// ---- BECKHOFF SPECIFIC helper library/POUs/MethodCall/UA_MethodCall_ADSReadWriteReq.TcPOU
FUNCTION_BLOCK UA_MethodCall_ADSReadWriteReq
VAR_INPUT
	bExecute			: BOOL;
	nConnectionHdl		: DWORD;
	nNamespaceIndex		: UINT; 			(* to be retrieved using UA_GetNamespaceIndex *)
	sNetID				: T_AmsNetId; 		(* AmsNetId OF the Target *)
	nPort				: INT; 			(* Port number	*)
	nIndexGroup			: DINT;			(* IndexGroup*)
	nIndexOffset		: DINT; 			(* IndexOffset*)
	pWriteData			: PVOID;
	cbWriteData			: UDINT;			(* Count of bytes to be read*)
	pReadArgInfoAndData	: PVOID;
	cbReadArgInfoAndData: UDINT;			(* Count of bytes to be read*)
	nNumberOfOutputArguments	: UDINT; 
	pOutputArgInfo		: POINTER TO ST_UAMethodArgInfo; 
	cbOutputArgInfo		: UDINT;
	Timeout				: TIME := DEFAULT_ADS_TIMEOUT;
END_VAR
VAR_OUTPUT
	cbReadData_R		: UDINT;
	bDone				: BOOL;
	bBusy				: BOOL;
	bError				: BOOL;
	nErrorID			: DWORD;
END_VAR
VAR
	iRdWrtReqState		: INT;
	RTrig				: R_TRIG;

	fbUA_MethodGetHandle: UA_MethodGetHandle;
	nMethodHdl			: DWORD;
	ObjectNodeID		: ST_UANodeID;
	MethodNodeID		: ST_UANodeID;

	fbUA_MethodCall		: UA_MethodCall;
	InputArguments		: ARRAY [1..nNumberOfInputArguments] OF ST_UAMethodArgInfo; (*ReadWriteReq has 6 input parameters *)	
	nArg				: INT;
	nInputData			: ARRAY [1..nInputArgSize] OF BYTE; // (* NetID(24)+ Port(2)+ IG(4)+ IO(4)*)
	nOffset				: UDINT;

	fbUA_MethodReleaseHandle	: UA_MethodReleaseHandle;
	bInputDataError				: BOOL; 
END_VAR
VAR CONSTANT
	nInputArgSize			: UDINT := 34; // (* NetID(24)+ Port(2)+ IG(4)+ IO(4)*)
	nNumberOfInputArguments : UDINT := 6;
END_VAR

(*
ADSReadWriteReq(
******** Input Arguments ********
	string sNetID, 		: AmsNetId of the Target
	int16 Port,			: Port number	
	int32 IndexGroup,		: IndexGroup
	int32 IndexOffset,		: IndexOffset
	ByteString WriteData	: Data to be written to the device
	uint32 cbReadData		: Count of bytes to be read
******** Output Arguments ********
	bytestring Data		: count of bytes actually read
);
*)

RTrig(CLK:= bExecute);

CASE iRdWrtReqState OF

0:	(* Get Method Handle *)
	IF RTrig.Q THEN
		bBusy		:= TRUE;
		bDone 		:= FALSE;
		bError		:= FALSE;
		nErrorID	:= 0;
		ObjectNodeID.eIdentifierType 	:= eUAIdentifierType_String;
		ObjectNodeID.nNamespaceIndex 	:= nNamespaceIndex;
		ObjectNodeID.sIdentifier		:= 'ADSAMS';
	
		MethodNodeID.eIdentifierType 	:= eUAIdentifierType_String;
		MethodNodeID.nNamespaceIndex 	:= nNamespaceIndex;
		MethodNodeID.sIdentifier		:= 'ADSAMS.AdsReadWriteReq';

		M_Init();
		IF bInputDataError = FALSE THEN
			iRdWrtReqState 	:= iRdWrtReqState + 1;
		ELSE
			bBusy		:= FALSE; 
			bError 		:= TRUE;
			nErrorID 	:= DEVICE_INVALIDSIZE; //16#705 parameter size not correct
		END_IF
	END_IF


1:	(* Method Get Handle *)
	fbUA_MethodGetHandle(
			Execute			:= TRUE,
			ConnectionHdl	:= nConnectionHdl,
			ObjectNodeID	:= ObjectNodeID,
			MethodNodeID 	:= MethodNodeID,
			Timeout			:= Timeout,
			MethodHdl		=> nMethodHdl
		);
	IF NOT fbUA_MethodGetHandle.Busy THEN
		fbUA_MethodGetHandle(Execute := FALSE);

		IF NOT fbUA_MethodGetHandle.Error THEN
			(*  *)
			iRdWrtReqState := iRdWrtReqState + 1; (* Call Method *)
		ELSE
			bError			:= TRUE;
			nErrorID		:= fbUA_MethodGetHandle.ErrorID;
			iRdWrtReqState := 3; (* Release Handle *)
		END_IF
	END_IF


2:	(* Method Call *)
	fbUA_MethodCall(
		Execute					:= TRUE,
		ConnectionHdl			:= nConnectionHdl,
		MethodHdl				:= nMethodHdl,
		nNumberOfInputArguments := nNumberOfInputArguments,		(* 6 *)
		pInputArgInfo			:= ADR(InputArguments),
		cbInputArgInfo			:= SIZEOF(InputArguments),
		pInputArgData			:= ADR(nInputData),
		cbInputArgData			:= nOffset,
		pInputWriteData			:= pWriteData,
		cbInputWriteData		:= cbWriteData,
		nNumberOfOutputArguments:= nNumberOfOutputArguments,		(* 6 *)
		pOutputArgInfo			:= pOutputArgInfo,
		cbOutputArgInfo			:= cbOutputArgInfo,
		pOutputArgInfoAndData	:= pReadArgInfoAndData,
		cbOutputArgInfoAndData	:= cbReadArgInfoAndData,
		Timeout					:= Timeout
	);
	IF NOT fbUA_MethodCall.Busy THEN
		fbUA_MethodCall(Execute := FALSE, cbRead_R => cbReadData_R);

		IF NOT fbUA_MethodCall.Error THEN
			(*  *)
			iRdWrtReqState 	:= iRdWrtReqState + 1; (* Release handle *)
		ELSE
			bError			:= TRUE;
			nErrorID		:= fbUA_MethodCall.ErrorID;
			iRdWrtReqState	:= 3; (* Release handle *)
		END_IF
	END_IF


3:	(* Release Method Handle *)
	fbUA_MethodReleaseHandle(
		Execute			:= TRUE,
		ConnectionHdl	:= nConnectionHdl,
		MethodHdl		:= nMethodHdl,
		Timeout			:= Timeout
	);

	IF NOT fbUA_MethodReleaseHandle.Busy THEN
		fbUA_MethodReleaseHandle(Execute := FALSE);
		bBusy := FALSE;
		IF NOT fbUA_MethodReleaseHandle.Error THEN
			(* session closed *)
			bDone := TRUE;
			iRdWrtReqState 	:= 0; (* idle *)
		ELSE
			bError		:= TRUE;
			nErrorID		:= fbUA_MethodReleaseHandle.ErrorID;
			iRdWrtReqState 	:= 0; (* idle *)
		END_IF
	END_IF
END_CASE

ACTION M_Init:
bInputDataError := FALSE; 
nOffset := 0;
MEMSET(ADR(InputArguments),0,SIZEOF(InputArguments));
MEMSET(ADR(nInputData),0,SIZEOF(nInputData));

nArg := 1;
(*sNetID := sAmsNetID;*)	(********** NET ID **********)
InputArguments[nArg].DataType			:= eUAType_String;
InputArguments[nArg].ValueRank			:= -1; 							(* Scalar = -1 or Array *)
InputArguments[nArg].ArrayDimensions[1]	:= 0; 							(* Number of Dimension in case its an array *)
InputArguments[nArg].nLenData			:= INT_TO_UDINT(LEN(sNetId)) + 1;				(* Length if its a STRING *)
IF nOffset + INT_TO_UDINT(LEN(sNetId))+1 > nInputArgSize THEN 
	bInputDataError := TRUE;
	RETURN;
ELSE
	MEMCPY(ADR(nInputData)+nOffset,ADR(sNetId),INT_TO_UDINT(LEN(sNetId))+1);				(* VALUE in BYTES FORM *)
	nOffset := nOffset + INT_TO_UDINT(LEN(sNetId))+1;
END_IF

nArg := nArg + 1;
(* nPort := 851;*)			(********** PORT **********)
InputArguments[nArg].DataType			:= eUAType_Int16;
InputArguments[nArg].ValueRank			:= -1; 							(* Scalar = -1 or Array *)
InputArguments[nArg].ArrayDimensions[1]	:= 0; 							(* Number of Dimension in case its an array *)
InputArguments[nArg].nLenData			:= SIZEOF(nPort);				(* Length if its a STRING *)
IF nOffset + SIZEOF(nPort) > nInputArgSize THEN 
	bInputDataError := TRUE;
	RETURN;
ELSE
	MEMCPY(ADR(nInputData)+nOffset,ADR(nPort),SIZEOF(nPort));			(* VALUE in BYTES FORM *)
	nOffset := nOffset + SIZEOF(nPort);
END_IF

nArg := nArg + 1;
(*nIndexGroup := 16#4020;*)	(********** INDEX GROUP **********)
InputArguments[nArg].DataType			:= eUAType_Int32;
InputArguments[nArg].ValueRank			:= -1; 							(* Scalar = -1 or Array *)
InputArguments[nArg].ArrayDimensions[1]	:= 0; 							(* Number of Dimension in case its an array *)
InputArguments[nArg].nLenData			:= SIZEOF(nIndexGroup);			(* Length if its a STRING *)
IF nOffset + SIZEOF(nIndexGroup) > nInputArgSize THEN 
	bInputDataError := TRUE;
	RETURN;
ELSE
	MEMCPY(ADR(nInputData)+nOffset,ADR(nIndexGroup),SIZEOF(nIndexGroup));		(* VALUE in BYTES FORM *)
	nOffset := nOffset + SIZEOF(nIndexGroup);
END_IF

nArg := nArg + 1;
(*nIndexOffset := 0; *)		(********** INDEX OFFSET **********)
InputArguments[nArg].DataType			:= eUAType_Int32;
InputArguments[nArg].ValueRank			:= -1; 							(* Scalar = -1 or Array *)
InputArguments[nArg].ArrayDimensions[1]	:= 0; 							(* Number of Dimension in case its an array *)
InputArguments[nArg].nLenData			:= SIZEOF(nIndexOffset);		(* Length if its a STRING *)
IF nOffset + SIZEOF(nIndexOffset) > nInputArgSize THEN 
	bInputDataError := TRUE;
	RETURN;
ELSE
	MEMCPY(ADR(nInputData)+nOffset,ADR(nIndexOffset),SIZEOF(nIndexOffset));	(* VALUE in BYTES FORM *)
	nOffset := nOffset + SIZEOF(nIndexOffset);
END_IF

nArg := nArg + 1;
(*Data := 2; *)		(*********** WriteData ***********)
InputArguments[nArg].DataType			:= eUAType_ByteString;
InputArguments[nArg].ValueRank			:= -1; 						(* Scalar = -1 or Array *)
InputArguments[nArg].ArrayDimensions[1]	:= 0; 						(* Number of Dimension in case its an array *)
InputArguments[nArg].nLenData			:= cbWriteData;				(* Length if its a STRING *)

nArg := nArg + 1;
(*Data := 2; *)		(*********** ReadData size ***********)
InputArguments[nArg].DataType			:= eUAType_UInt32;
InputArguments[nArg].ValueRank			:= -1; 						(* Scalar = -1 or Array *)
InputArguments[nArg].ArrayDimensions[1]	:= 0; 						(* Number of Dimension in case its an array *)
InputArguments[nArg].nLenData			:= SIZEOF(cbReadArgInfoAndData);		(* Length if its a STRING *)
END_ACTION

END_FUNCTION_BLOCK

// ---- POUs/PRG_READ_List_woConnectIdent.TcPOU
PROGRAM PRG_READ_List_woConnectIdent
VAR
	fbUA_Connect			: UA_Connect;
	SessionConnectInfo		: ST_UASessionConnectInfo;
	sOpcUA_URL				: STRING(MAX_STRING_LENGTH);
	nConnectionHdl			: DWORD;

	fbUA_GetNamespaceIndex 	: UA_GetNamespaceIndex;
	nNamespaceIndex			: UINT;
	fbUA_NodeGetHandleList	: UA_NodeGetHandleList;
	NodeIDs					: ARRAY [1..nMaxNodeIDsInList] OF ST_UANodeID;
	nNodeHdls				: ARRAY [1..nMaxNodeIDsInList] OF DWORD;

	fbUA_ReadList			: UA_ReadList; 
	stIndexRange			: ARRAY [1..nMaxIndexRange] OF ST_UAIndexRange;
	nIndexRangeCount		: UINT;
	stNodeAddInfo			: ARRAY [1..nMaxNodeIDsInList] OF ST_UANodeAdditionalInfo;
	stReadListData			: ST_ReadListData; // memory block must contain the Data[], NodeErrorIDs[], TimeStamps[] and cbData_R[]
	cbData					: ARRAY [1..nMaxNodeIDsInList] OF UDINT; (* Bytes to be actually Read *)
	cbData_R				: UDINT;
	cbDataTotal				: UDINT; 
	
	fbUA_NodeReleaseHandleList	: UA_NodeReleaseHandleList;

	fbUA_Disconnect		: UA_Disconnect;

	iState		: INT;
	bTest		: BOOL:= TRUE;
	bDone		: BOOL;
	bBusy		: BOOL;
	bError		: BOOL;
	nErrorID	: DWORD;
	
	nNodeIdx	: INT; 
END_VAR


CASE iState OF
0:	(* idle *)
	IF bTest THEN
		bTest		:= FALSE;
		bError		:= FALSE;
		nErrorID	:= 0;

		(* Parameterize *)
		sOpcUA_URL						:= 'opc.tcp://pujal-nb03:4840';	(* OpcUA Url of the device with ip address *)

		SessionConnectInfo.tConnectTimeout 		:= T#1S;
		SessionConnectInfo.tSessionTimeout 		:= T#1S;
		SessionConnectInfo.sApplicationName		:= '';
//		SessionConnectInfo.sApplicationUri 		:= '';
		SessionConnectInfo.eSecurityMode 		:= eUASecurityMsgMode_None;
		SessionConnectInfo.eSecurityPolicyUri 	:= eUASecurityPolicy_None;
		SessionConnectInfo.eTransportProfileUri := eUATransportProfileUri_UATcp;

(*		nIndexRange[1].nStartIndex := 0;
		nIndexRange[1].nEndIndex := 1;
		nIndexRange[1].bRangeAccess := TRUE; *)
		iState	:= iState + 1;
	END_IF

1:	(* open UA session *)
	fbUA_Connect(
		Execute				:= TRUE,
		ServerURL			:= sOpcUA_URL,
		SessionConnectInfo  := SessionConnectInfo,
		Timeout				:= T#5S,
		ConnectionHdl		=> nConnectionHdl
	);

	IF NOT fbUA_Connect.Busy THEN
		fbUA_Connect(Execute := FALSE);

		IF NOT fbUA_Connect.Error THEN
			(* session open *)
			iState := iState + 1;
		ELSE
			bError			:= TRUE;
			nErrorID		:= fbUA_Connect.ErrorID;
			nConnectionHdl	:= 0;
			iState 			:= 0; (* idle *)
		END_IF
	END_IF


2:	(* GetNS Index *)
	fbUA_GetNamespaceIndex(
		Execute			:= TRUE,
		ConnectionHdl	:= nConnectionHdl,
		NamespaceUri	:= 'PLC1',
		NamespaceIndex	=> nNamespaceIndex
	);

	IF NOT fbUA_GetNamespaceIndex.Busy THEN
		fbUA_GetNamespaceIndex(Execute := FALSE);
		IF NOT fbUA_GetNamespaceIndex.Error THEN
			(* session closed *)
			iState 		:= iState + 1; (* idle *)
		ELSE
			bError		:= TRUE;
			nErrorID	:= fbUA_GetNamespaceIndex.ErrorID;
			iState 		:= 6; (* idle *)
		END_IF
	END_IF


3:	(* Get Node Handle *)
//	stNodeAddInfo[1].nIndexRangeCount := nIndexRangeCount;
//	stNodeAddInfo[1].stIndexRange := stIndexRange;
//	stNodeAddInfo[2].nIndexRangeCount := nIndexRangeCount;
//	stNodeAddInfo[2].stIndexRange := stIndexRange;
	nNodeIdx := 1;		//1
	
	NodeIDs[nNodeIdx].eIdentifierType := eUAIdentifierType_String;
	NodeIDs[nNodeIdx].nNamespaceIndex := nNamespaceIndex;
	NodeIDs[nNodeIdx].sIdentifier	:= 'MAIN.iVar1';
	
	nNodeIdx := nNodeIdx + 1; //2
	NodeIDs[nNodeIdx].eIdentifierType := eUAIdentifierType_String;
	NodeIDs[nNodeIdx].nNamespaceIndex := nNamespaceIndex;
	NodeIDs[nNodeIdx].sIdentifier	:= 'MAIN.diVar1';
	
	nNodeIdx := nNodeIdx + 1; //3
	NodeIDs[nNodeIdx].eIdentifierType := eUAIdentifierType_String;
	NodeIDs[nNodeIdx].nNamespaceIndex := nNamespaceIndex;
	NodeIDs[nNodeIdx].sIdentifier	:= 'MAIN.iVar2';
	
	nNodeIdx := nNodeIdx + 1; //4
	NodeIDs[nNodeIdx].eIdentifierType := eUAIdentifierType_String;
	NodeIDs[nNodeIdx].nNamespaceIndex := nNamespaceIndex;
	NodeIDs[nNodeIdx].sIdentifier	:= 'MAIN.diVar2';

	fbUA_NodeGetHandleList(
		Execute			:= TRUE,
		ConnectionHdl	:= nConnectionHdl,
		NodeIDCount 	:= gNodeIDCount, // 4
		NodeIDs			:= NodeIDs,
		NodeHdls		=> nNodeHdls
	);

	IF NOT fbUA_NodeGetHandleList.Busy THEN
		fbUA_NodeGetHandleList(Execute := FALSE);

		IF NOT fbUA_NodeGetHandleList.Error THEN
			(* session closed *)
			iState 		:= iState + 1; (* idle *)
		ELSE
			bError		:= TRUE;
			nErrorID	:= fbUA_NodeGetHandleList.ErrorID;
			iState 		:= 6; (* idle *)
		END_IF
	END_IF

	
4: 	(* UA_Read *)
	cbData[1] := SIZEOF(stReadListData.nIntVar1);
	cbData[2] := SIZEOF(stReadListData.nIntVar2);
	cbData[3] := SIZEOF(stReadListData.nIntVar3);
	cbData[4] := SIZEOF(stReadListData.nIntVar4);
	cbDataTotal := SIZEOF(stReadListData);
	fbUA_ReadList(
		Execute			:= TRUE,
		ConnectionHdl	:= nConnectionHdl,
		NodeHdlCount	:= gNodeIDCount, // 4
		NodeHdls		:= nNodeHdls,
		stNodeAddInfo 	:= stNodeAddInfo,
		pVariable		:= ADR(stReadListData),
		cbData			:= cbData ,
		cbDataTotal		:= cbDataTotal		
		);

	IF NOT fbUA_ReadList.Busy THEN
		fbUA_ReadList( Execute := FALSE, cbData_R => cbData_R);

		IF NOT fbUA_ReadList.Error THEN
			(* session closed *)
			iState 		:= iState + 1; (* idle *)
		ELSE
			bError		:= TRUE;
			nErrorID	:= fbUA_ReadList.ErrorID;
			iState 		:= 6; (* idle *)
		END_IF
	END_IF


5:	(* Release Node Handle *)
	fbUA_NodeReleaseHandleList(
		Execute			:= TRUE,
		ConnectionHdl	:= nConnectionHdl,
		NodeHdlCount	:= gNodeIDCount,	// 4
		NodeHdls		:= nNodeHdls
	);

	IF NOT fbUA_NodeReleaseHandleList.Busy THEN
		fbUA_NodeReleaseHandleList(Execute := FALSE);

		IF NOT fbUA_NodeReleaseHandleList.Error THEN
			(* session closed *)
			iState 		:= iState + 1; (* idle *)
		ELSE
			bError		:= TRUE;
			nErrorID	:= fbUA_NodeReleaseHandleList.ErrorID;
			iState 		:= 6; (* idle *)
		END_IF
	END_IF


6:	(* close session *)
	fbUA_Disconnect(
		Execute			:= TRUE,
		ConnectionHdl	:= nConnectionHdl
	);

	IF NOT fbUA_Disconnect.Busy THEN
		fbUA_Disconnect(Execute := FALSE);
		bBusy := FALSE;
		IF NOT fbUA_Disconnect.Error THEN
			(* session closed *)
			iState 		:= 0; (* idle *)
			IF NOT bError THEN 
				bDone 	:= TRUE;
			END_IF
		ELSE
			bError			:= TRUE;
			nErrorID		:= fbUA_Disconnect.ErrorID;
			iState 			:= 0; (* idle *)
			nConnectionHdl	:= 0;
		END_IF
	END_IF
END_CASE

END_PROGRAM

// ---- POUs/PRG_READ_List.TcPOU
PROGRAM PRG_READ_List
VAR
	fbUA_ConnectEx			: UA_Connect;
	SessionConnectInfoEx	: ST_UASessionConnectInfo;
	sOpcUA_URL				: STRING(MAX_STRING_LENGTH);
	nConnectionHdl			: DWORD;

	fbUA_GetNamespaceIndex 	: UA_GetNamespaceIndex;
	nNamespaceIndex			: UINT;
	fbUA_NodeGetHandleList	: UA_NodeGetHandleList;
	
	NodeIDs					: ARRAY [1..nMaxNodeIDsInList] OF ST_UANodeID;
	nNodeHdls				: ARRAY [1..nMaxNodeIDsInList] OF DWORD;

	fbUA_ReadList			: UA_ReadList;
	stIndexRange			: ARRAY [1..nMaxIndexRange] OF ST_UAIndexRange;
	nIndexRangeCount		: UINT;
	stNodeAddInfo			: ARRAY [1..nMaxNodeIDsInList] OF ST_UANodeAdditionalInfo;
	stReadListData			: ST_ReadListData; // memory block must contain the Data[], NodeErrorIDs[], TimeStamps[] and cbData_R[]
	cbData					: ARRAY [1..nMaxNodeIDsInList] OF UDINT; (* Bytes to be actually Read *)
	cbData_R				: UDINT;
	cbDataTotal				: UDINT; 
	
	fbUA_NodeReleaseHandleList	: UA_NodeReleaseHandleList;

	fbUA_Disconnect		: UA_Disconnect;

	iState		: INT;
	bTest		: BOOL:= TRUE;
	bDone		: BOOL;
	bBusy		: BOOL;
	bError		: BOOL;
	nErrorID	: DWORD;
	
	nNodeIdx	: INT; 
END_VAR


CASE iState OF
0:	(* idle *)
	IF bTest THEN
		bTest		:= FALSE;
		bError		:= FALSE;
		nErrorID	:= 0;

		(* Parameterize *)
		sOpcUA_URL						:= 'opc.tcp://pujal-nb03:4840';	(* OpcUA Url of the device with ip address *)

		SessionConnectInfoEx.tConnectTimeout 		:= T#5S;
		SessionConnectInfoEx.tSessionTimeout 		:= T#5S;
		SessionConnectInfoEx.sApplicationName		:= '';
		SessionConnectInfoEx.eSecurityMode 			:= eUASecurityMsgMode_None;
		SessionConnectInfoEx.eSecurityPolicyUri 	:= eUASecurityPolicy_None;
		SessionConnectInfoEx.eTransportProfileUri 	:= eUATransportProfileUri_UATcp;
		//SessionConnectInfoEx.stUserIdentTokenType

(*		nIndexRange[1].nStartIndex := 0;
		nIndexRange[1].nEndIndex := 1;
		nIndexRange[1].bRangeAccess := TRUE; *)
		iState	:= iState + 1;
	END_IF

1:	(* open UA session *)
	fbUA_ConnectEx(
		Execute				:= TRUE,
		ServerURL			:= sOpcUA_URL,
		SessionConnectInfo	:= SessionConnectInfoEx,
		Timeout				:= T#5S,
		ConnectionHdl		=> nConnectionHdl
	);

	IF NOT fbUA_ConnectEx.Busy THEN
		fbUA_ConnectEx(Execute := FALSE);

		IF NOT fbUA_ConnectEx.Error THEN
			(* session open *)
			iState := iState + 1;
		ELSE
			bError			:= TRUE;
			nErrorID		:= fbUA_ConnectEx.ErrorID;
			nConnectionHdl	:= 0;
			iState 			:= 0; (* idle *)
		END_IF
	END_IF


2:	(* GetNS Index *)
	fbUA_GetNamespaceIndex(
		Execute			:= TRUE,
		ConnectionHdl	:= nConnectionHdl,
		NamespaceUri	:= 'PLC1',
		NamespaceIndex	=> nNamespaceIndex
	);

	IF NOT fbUA_GetNamespaceIndex.Busy THEN
		fbUA_GetNamespaceIndex(Execute := FALSE);
		IF NOT fbUA_GetNamespaceIndex.Error THEN
			(* session closed *)
			iState 		:= iState + 1; (* idle *)
		ELSE
			bError		:= TRUE;
			nErrorID	:= fbUA_GetNamespaceIndex.ErrorID;
			iState 		:= 6; (* idle *)
		END_IF
	END_IF


3:	(* Get Node Handle *)
	nNodeIdx := 1;	
	NodeIDs[nNodeIdx].eIdentifierType := eUAIdentifierType_String;
	NodeIDs[nNodeIdx].nNamespaceIndex := nNamespaceIndex;
	NodeIDs[nNodeIdx].sIdentifier	:= 'MAIN.iVar1';
	cbData[nNodeIdx] := SIZEOF(stReadListData.nIntVar1);
	
	nNodeIdx := nNodeIdx + 1; 
	NodeIDs[nNodeIdx].eIdentifierType := eUAIdentifierType_String;
	NodeIDs[nNodeIdx].nNamespaceIndex := nNamespaceIndex;
	NodeIDs[nNodeIdx].sIdentifier	:= 'MAIN.iVar2';
	cbData[nNodeIdx] := SIZEOF(stReadListData.nIntVar2);
	
	nNodeIdx := nNodeIdx + 1; 	
	NodeIDs[nNodeIdx].eIdentifierType := eUAIdentifierType_String;
	NodeIDs[nNodeIdx].nNamespaceIndex := nNamespaceIndex;
	NodeIDs[nNodeIdx].sIdentifier	:= 'MAIN.iVar1';	
	cbData[nNodeIdx] := SIZEOF(stReadListData.nIntVar3);
	
	nNodeIdx := nNodeIdx + 1; 
	NodeIDs[nNodeIdx].eIdentifierType := eUAIdentifierType_String;
	NodeIDs[nNodeIdx].nNamespaceIndex := nNamespaceIndex;
	NodeIDs[nNodeIdx].sIdentifier	:= 'MAIN.iVar1';	
	cbData[nNodeIdx] := SIZEOF(stReadListData.nIntVar4);
	
	nNodeIdx := nNodeIdx + 1; 
	NodeIDs[nNodeIdx].eIdentifierType := eUAIdentifierType_String;
	NodeIDs[nNodeIdx].nNamespaceIndex := nNamespaceIndex;
	NodeIDs[nNodeIdx].sIdentifier	:= 'MAIN.iVar1';	
	cbData[nNodeIdx] := SIZEOF(stReadListData.nIntVar5);

	nNodeIdx := nNodeIdx + 1; 
	NodeIDs[nNodeIdx].eIdentifierType := eUAIdentifierType_String;
	NodeIDs[nNodeIdx].nNamespaceIndex := nNamespaceIndex;
	NodeIDs[nNodeIdx].sIdentifier	:= 'MAIN.iVar1';	
	cbData[nNodeIdx] := SIZEOF(stReadListData.nIntVar6);

	nNodeIdx := nNodeIdx + 1; 
	NodeIDs[nNodeIdx].eIdentifierType := eUAIdentifierType_String;
	NodeIDs[nNodeIdx].nNamespaceIndex := nNamespaceIndex;
	NodeIDs[nNodeIdx].sIdentifier	:= 'MAIN.iVar1';	
	cbData[nNodeIdx] := SIZEOF(stReadListData.nIntVar7);

	nNodeIdx := nNodeIdx + 1; 
	NodeIDs[nNodeIdx].eIdentifierType := eUAIdentifierType_String;
	NodeIDs[nNodeIdx].nNamespaceIndex := nNamespaceIndex;
	NodeIDs[nNodeIdx].sIdentifier	:= 'MAIN.iVar1';
	cbData[nNodeIdx] := SIZEOF(stReadListData.nIntVar8);	

	nNodeIdx := nNodeIdx + 1; 
	NodeIDs[nNodeIdx].eIdentifierType := eUAIdentifierType_String;
	NodeIDs[nNodeIdx].nNamespaceIndex := nNamespaceIndex;
	NodeIDs[nNodeIdx].sIdentifier	:= 'MAIN.iVar1';
	cbData[nNodeIdx] := SIZEOF(stReadListData.nIntVar9);

	nNodeIdx := nNodeIdx + 1; 
	NodeIDs[nNodeIdx].eIdentifierType := eUAIdentifierType_String;
	NodeIDs[nNodeIdx].nNamespaceIndex := nNamespaceIndex;
	NodeIDs[nNodeIdx].sIdentifier	:= 'MAIN.iVar1';
	cbData[nNodeIdx] := SIZEOF(stReadListData.nIntVar10);	

	cbDataTotal := SIZEOF(stReadListData);
	
	fbUA_NodeGetHandleList(
		Execute			:= TRUE,
		ConnectionHdl	:= nConnectionHdl,
		NodeIDCount 	:= gNodeIDCount, // 10
		NodeIDs			:= NodeIDs,
		NodeHdls		=> nNodeHdls
	);

	IF NOT fbUA_NodeGetHandleList.Busy THEN
		fbUA_NodeGetHandleList(Execute := FALSE);

		IF NOT fbUA_NodeGetHandleList.Error THEN
			(* session closed *)
			iState 		:= iState + 1; (* idle *)
		ELSE
			bError		:= TRUE;
			nErrorID	:= fbUA_NodeGetHandleList.ErrorID;
			iState 		:= 6; (* idle *)
		END_IF
	END_IF

	
4: 	(* UA_Read *)
	
	fbUA_ReadList(
		Execute			:= TRUE,
		ConnectionHdl	:= nConnectionHdl,
		NodeHdlCount	:= gNodeIDCount, // 2
		NodeHdls		:= nNodeHdls,
		stNodeAddInfo 	:= stNodeAddInfo,
		pVariable		:= ADR(stReadListData),
		cbData			:= cbData ,
		cbDataTotal		:= cbDataTotal		
		);

	IF NOT fbUA_ReadList.Busy THEN
		fbUA_ReadList( Execute := FALSE, cbData_R => cbData_R);

		IF NOT fbUA_ReadList.Error THEN
			(* session closed *)
			iState 		:= iState + 1; (* idle *)
		ELSE
			bError		:= TRUE;
			nErrorID	:= fbUA_ReadList.ErrorID;
			iState 		:= 6; (* idle *)
		END_IF
	END_IF


5:	(* Release Node Handle *)
	fbUA_NodeReleaseHandleList(
		Execute			:= TRUE,
		ConnectionHdl	:= nConnectionHdl,
		NodeHdlCount	:= gNodeIDCount,
		NodeHdls		:= nNodeHdls
	);

	IF NOT fbUA_NodeReleaseHandleList.Busy THEN
		fbUA_NodeReleaseHandleList(Execute := FALSE);

		IF NOT fbUA_NodeReleaseHandleList.Error THEN
			(* session closed *)
			iState 		:= iState + 1; (* idle *)
		ELSE
			bError		:= TRUE;
			nErrorID	:= fbUA_NodeReleaseHandleList.ErrorID;
			iState 		:= 6; (* idle *)
		END_IF
	END_IF


6:	(* close session *)
	fbUA_Disconnect(
		Execute			:= TRUE,
		ConnectionHdl	:= nConnectionHdl
	);

	IF NOT fbUA_Disconnect.Busy THEN
		fbUA_Disconnect(Execute := FALSE);
		bBusy := FALSE;
		IF NOT fbUA_Disconnect.Error THEN
			(* session closed *)
			iState 		:= 0; (* idle *)
			IF NOT bError THEN 
				bDone 	:= TRUE;
			END_IF
		ELSE
			bError			:= TRUE;
			nErrorID		:= fbUA_Disconnect.ErrorID;
			iState 			:= 0; (* idle *)
			nConnectionHdl	:= 0;
		END_IF
	END_IF
END_CASE

END_PROGRAM

// ---- POUs/PRG_READ_List_ArrayInt.TcPOU
PROGRAM PRG_READ_List_ArrayInt
VAR
	fbUA_Connect			: UA_Connect;
	SessionConnectInfo		: ST_UASessionConnectInfo;
	sOpcUA_URL				: STRING(MAX_STRING_LENGTH);
	nConnectionHdl			: DWORD;

	fbUA_GetNamespaceIndex 	: UA_GetNamespaceIndex;
	nNamespaceIndex			: UINT;
	fbUA_NodeGetHandleList	: UA_NodeGetHandleList;
	NodeIDs					: ARRAY [1..nMaxNodeIDsInList] OF ST_UANodeID;
	nNodeHdls				: ARRAY [1..nMaxNodeIDsInList] OF DWORD;

	fbUA_ReadList			: UA_ReadList; 
	stIndexRange			: ARRAY [1..nMaxIndexRange] OF ST_UAIndexRange;
	nIndexRangeCount		: UINT;
	stNodeAddInfo			: ARRAY [1..nMaxNodeIDsInList] OF ST_UANodeAdditionalInfo;
	stReadListDataArrayInt	: ST_ReadListDataArrayInt; // memory block must contain the Data[], NodeErrorIDs[], TimeStamps[] and cbData_R[]
	cbData					: ARRAY [1..nMaxNodeIDsInList] OF UDINT; (* Bytes to be actually Read *)
	cbData_R				: UDINT;
	cbDataTotal				: UDINT; 
	
	fbUA_NodeReleaseHandleList	: UA_NodeReleaseHandleList;

	fbUA_Disconnect		: UA_Disconnect;

	iState		: INT;
	bTest		: BOOL:= TRUE;
	bDone		: BOOL;
	bBusy		: BOOL;
	bError		: BOOL;
	nErrorID	: DWORD;
	
	nNodeIdx	: INT; 
END_VAR


CASE iState OF
0:	(* idle *)
	IF bTest THEN
		bTest		:= FALSE;
		bError		:= FALSE;
		nErrorID	:= 0;

		(* Parameterize *)
		sOpcUA_URL						:= 'opc.tcp://pujal-nb03:4840';	(* OpcUA Url of the device with ip address *)

		SessionConnectInfo.tConnectTimeout 		:= T#1S;
		SessionConnectInfo.tSessionTimeout 		:= T#1S;
		SessionConnectInfo.sApplicationName		:= '';
//		SessionConnectInfo.sApplicationUri 		:= '';
		SessionConnectInfo.eSecurityMode 		:= eUASecurityMsgMode_None;
		SessionConnectInfo.eSecurityPolicyUri 	:= eUASecurityPolicy_None;
		SessionConnectInfo.eTransportProfileUri := eUATransportProfileUri_UATcp;

(*		nIndexRange[1].nStartIndex := 0;
		nIndexRange[1].nEndIndex := 1;
		nIndexRange[1].bRangeAccess := TRUE; *)
		iState	:= iState + 1;
	END_IF

1:	(* open UA session *)
	fbUA_Connect(
		Execute				:= TRUE,
		ServerURL			:= sOpcUA_URL,
		SessionConnectInfo  := SessionConnectInfo,
		Timeout				:= T#5S,
		ConnectionHdl		=> nConnectionHdl
	);

	IF NOT fbUA_Connect.Busy THEN
		fbUA_Connect(Execute := FALSE);

		IF NOT fbUA_Connect.Error THEN
			(* session open *)
			iState := iState + 1;
		ELSE
			bError			:= TRUE;
			nErrorID		:= fbUA_Connect.ErrorID;
			nConnectionHdl	:= 0;
			iState 			:= 0; (* idle *)
		END_IF
	END_IF


2:	(* GetNS Index *)
	fbUA_GetNamespaceIndex(
		Execute			:= TRUE,
		ConnectionHdl	:= nConnectionHdl,
		NamespaceUri	:= 'PLC1',
		NamespaceIndex	=> nNamespaceIndex
	);

	IF NOT fbUA_GetNamespaceIndex.Busy THEN
		fbUA_GetNamespaceIndex(Execute := FALSE);
		IF NOT fbUA_GetNamespaceIndex.Error THEN
			(* session closed *)
			iState 		:= iState + 1; (* idle *)
		ELSE
			bError		:= TRUE;
			nErrorID	:= fbUA_GetNamespaceIndex.ErrorID;
			iState 		:= 6; (* idle *)
		END_IF
	END_IF


3:	(* Get Node Handle *)
//	stNodeAddInfo[1].nIndexRangeCount := nIndexRangeCount;
//	stNodeAddInfo[1].stIndexRange := stIndexRange;
//	stNodeAddInfo[2].nIndexRangeCount := nIndexRangeCount;
//	stNodeAddInfo[2].stIndexRange := stIndexRange;
	nNodeIdx := 1;		//1
	
	NodeIDs[nNodeIdx].eIdentifierType := eUAIdentifierType_String;
	NodeIDs[nNodeIdx].nNamespaceIndex := nNamespaceIndex;
	NodeIDs[nNodeIdx].sIdentifier	:= 'MAIN.iArrayIntVar1';
	
	nNodeIdx := nNodeIdx + 1; //2
	NodeIDs[nNodeIdx].eIdentifierType := eUAIdentifierType_String;
	NodeIDs[nNodeIdx].nNamespaceIndex := nNamespaceIndex;
	NodeIDs[nNodeIdx].sIdentifier	:= 'MAIN.diArrayDintVar2';

	fbUA_NodeGetHandleList(
		Execute			:= TRUE,
		ConnectionHdl	:= nConnectionHdl,
		NodeIDCount 	:= gNodeIDCount_Array, // 2
		NodeIDs			:= NodeIDs,
		NodeHdls		=> nNodeHdls
	);

	IF NOT fbUA_NodeGetHandleList.Busy THEN
		fbUA_NodeGetHandleList(Execute := FALSE);

		IF NOT fbUA_NodeGetHandleList.Error THEN
			(* session closed *)
			iState 		:= iState + 1; (* idle *)
		ELSE
			bError		:= TRUE;
			nErrorID	:= fbUA_NodeGetHandleList.ErrorID;
			iState 		:= 6; (* idle *)
		END_IF
	END_IF

	
4: 	(* UA_Read *)
	cbData[1] := SIZEOF(stReadListDataArrayInt.nArrIntVar1);
	cbData[2] := SIZEOF(stReadListDataArrayInt.nArrDintVar2);

	cbDataTotal := SIZEOF(stReadListDataArrayInt);
	fbUA_ReadList(
		Execute			:= TRUE,
		ConnectionHdl	:= nConnectionHdl,
		NodeHdlCount	:= gNodeIDCount_Array, // 2
		NodeHdls		:= nNodeHdls,
		stNodeAddInfo 	:= stNodeAddInfo,
		pVariable		:= ADR(stReadListDataArrayInt),
		cbData			:= cbData ,
		cbDataTotal		:= cbDataTotal		
		);

	IF NOT fbUA_ReadList.Busy THEN
		fbUA_ReadList( Execute := FALSE, cbData_R => cbData_R);

		IF NOT fbUA_ReadList.Error THEN
			(* session closed *)
			iState 		:= iState + 1; (* idle *)
		ELSE
			bError		:= TRUE;
			nErrorID	:= fbUA_ReadList.ErrorID;
			iState 		:= 6; (* idle *)
		END_IF
	END_IF


5:	(* Release Node Handle *)
	fbUA_NodeReleaseHandleList(
		Execute			:= TRUE,
		ConnectionHdl	:= nConnectionHdl,
		NodeHdlCount	:= gNodeIDCount_Array,
		NodeHdls		:= nNodeHdls
	);

	IF NOT fbUA_NodeReleaseHandleList.Busy THEN
		fbUA_NodeReleaseHandleList(Execute := FALSE);

		IF NOT fbUA_NodeReleaseHandleList.Error THEN
			(* session closed *)
			iState 		:= iState + 1; (* idle *)
		ELSE
			bError		:= TRUE;
			nErrorID	:= fbUA_NodeReleaseHandleList.ErrorID;
			iState 		:= 6; (* idle *)
		END_IF
	END_IF


6:	(* close session *)
	fbUA_Disconnect(
		Execute			:= TRUE,
		ConnectionHdl	:= nConnectionHdl
	);

	IF NOT fbUA_Disconnect.Busy THEN
		fbUA_Disconnect(Execute := FALSE);
		bBusy := FALSE;
		IF NOT fbUA_Disconnect.Error THEN
			(* session closed *)
			iState 		:= 0; (* idle *)
			IF NOT bError THEN 
				bDone 	:= TRUE;
			END_IF
		ELSE
			bError			:= TRUE;
			nErrorID		:= fbUA_Disconnect.ErrorID;
			iState 			:= 0; (* idle *)
			nConnectionHdl	:= 0;
		END_IF
	END_IF
END_CASE

END_PROGRAM

// ---- Test_CloudSample/POUs/CloudSample_SQL.TcPOU
PROGRAM CloudSample_SQL
VAR
	(* Declarations for Cloud connect to Microsoft Azure Cloud *)
	bInsertAzure					: BOOL;
	bInsertAzureCyclic				: BOOL;
	nStateAzure						: BYTE := 0;
	R_TRIGAzure						: R_TRIG;
	
	ObjectNodeID					: ST_UANodeID;
	MethodNodeID					: ST_UANodeID;

	bErrorAzure						: BOOL; 
	nErrorIDAzure					: DWORD;
				
	fb_OpcUAConnectAzure			: UA_Connect;
	SessionConnectInfo				: ST_UASessionConnectInfo;
	sOpcUA_URLAzure					: STRING(MAX_STRING_LENGTH);
	hUAConnectionHdlAzure			: UDINT;
	
	fbUA_OpcUAGetNSIndexAzure 		: UA_GetNamespaceIndex;
	nNamespaceIndexAzure			: UINT;
	
	fbMethodCall_DBRecordInsert		: UA_MethodCall_DBRecordInsert;
	stUASQLState					: ST_UASQLState;
	
	fbBuildSqlInsertAzure			: FB_BuildSQLInsert;
	sSqlInsertAzure					: STRING(100);	
	
	fb_OpcUADisconnectAzure			: UA_Disconnect;
	bUADisconnectStartAzure			: BOOL; 
	
	(* Miscellaneous variables *)
	fbRandom					: DRAND;
	lrRandom					: LREAL;
	sRandom						: STRING(MAX_DATA_ACCURACY);
	sRandom2					: STRING(MAX_DATA_ACCURACY);
	fbNTGetTime					: NT_GetTime;
	bBusyTime					: BOOL;
	stTime						: TIMESTRUCT;
	
	bInit			: BOOL := TRUE;
END_VAR

(* Create random number for upload into the Cloud *)
fbRandom(
	Seed := 1,
	Num => lrRandom);
lrRandom := lrRandom * 10;
sRandom := LREAL_TO_STRING(lrRandom);

(* The value of Poti 1 will be used to write into Cloud *)
sRandom2 := INT_TO_STRING(us_Poti_1);
IF bInit THEN 
	M_Init();
	bInit := FALSE; 
END_IF
R_TRIGAzure(CLK := bInsertAzure);
(* Upload once to Microsoft Azure Cloud *)
CASE nStateAzure OF
	0:
	 	(* To start this sample you have to set a rising edge to the variable bInsertAzure *)
		IF R_TRIGAzure.Q OR bInsertAzureCyclic THEN
			M_Init();
			nStateAzure 	:= 1;		
			bInsertAzure 	:= FALSE;
			bInsertAzureCyclic := TRUE;
			bErrorAzure 	:= FALSE; 
			nErrorIDAzure 	:= 0; 
		END_IF
			
	1:
		(* Get System Time to create timestamp*)
		fbNTGetTime(
			NETID 	:= '',
			START	:= TRUE,
			TMOUT 	:= T#5S,
			BUSY 	=> bBusyTime,
			TIMESTR => stTime);
		
		IF NOT bBusyTime THEN
			fbNTGetTime(START := FALSE);
			nStateAzure := 2;
		END_IF

	2:
		(* Establish session to OPC-UA Server *)
		IF hUAConnectionHdlAzure = 0 THEN
			fb_OpcUAConnectAzure(
				Execute 			:= TRUE,
				ServerUrl 			:= 'opc.tcp://ew2013vm.cloudapp.net:4840',
				SessionConnectInfo 	:= SessionConnectInfo,
				Timeout 			:= T#5S,
				ConnectionHdl 		=> hUAConnectionHdlAzure
				);
		ELSE
			nStateAzure := 4; 		
		END_IF
		
		IF NOT fb_OpcUAConnectAzure.Busy THEN
			fb_OpcUAConnectAzure(Execute := FALSE);
			IF NOT fb_OpcUAConnectAzure.Error THEN
				nStateAzure := 3;
			ELSE
				(* Error Occurred *)
				bErrorAzure	 := TRUE; 
				nErrorIDAzure := fb_OpcUAConnectAzure.ErrorID;
			END_IF	
		END_IF	
		
	3: 
		(* GetNS Index *)
		fbUA_OpcUAGetNSIndexAzure(
			Execute			:= TRUE,
			ConnectionHdl	:= hUAConnectionHdlAzure,
			NamespaceUri	:= 'ADSAMS',
			NamespaceIndex	=> nNamespaceIndexAzure
		);
	
		IF NOT fbUA_OpcUAGetNSIndexAzure.Busy THEN
			fbUA_OpcUAGetNSIndexAzure(Execute := FALSE);
			IF NOT fbUA_OpcUAGetNSIndexAzure.Error THEN
				(* session closed *)
				ObjectNodeID.eIdentifierType := eUAIdentifierType_String;
				ObjectNodeID.nNamespaceIndex := nNamespaceIndexAzure;
				ObjectNodeID.sIdentifier	 := 'ADSAMS';
				
				MethodNodeID.eIdentifierType := eUAIdentifierType_String;
				MethodNodeID.nNamespaceIndex := nNamespaceIndexAzure;
				MethodNodeID.sIdentifier	 := 'ADSAMS.AdsReadWriteReq';
				nStateAzure := 4; (* method *)
			ELSE
				(* Error occurred *)
				bErrorAzure	 := TRUE; 
				nErrorIDAzure := fbUA_OpcUAGetNSIndexAzure.ErrorID;
			END_IF
		END_IF
	
	4:
		 (* Prepare SQL Insert for Cloud *)
		fbBuildSqlInsertAzure(
			sTableName 		:= 'Zaehlerdaten',
			stTimestamp 	:= stTime,
			uiMesstellenID 	:= 2,
			stLogger 		:= 'HelloWorld',
			rMesswert 		:= 42,
			stEinheit 		:= 'Celsius',
			sValue 			:= sRandom2,
			sQuery 			=> sSqlInsertAzure);
		
		(* Write data to the Microsoft Azure cloud via OPC-UA *)
		fbMethodCall_DBRecordInsert(
			bExecute		:= TRUE, 
			nConnectionHdl	:= hUAConnectionHdlAzure, 
			nNamespaceIndex	:= nNamespaceIndexAzure, 
			pWriteData		:= ADR(sSqlInsertAzure), 
			cbWriteData		:= INT_TO_UDINT(LEN(sSqlInsertAzure))+1, 
			stUASQLState	=> stUASQLState);

		
		IF NOT fbMethodCall_DBRecordInsert.bBusy THEN
			fbMethodCall_DBRecordInsert(bExecute := FALSE,stUASQLState	=> stUASQLState);
			IF NOT fbMethodCall_DBRecordInsert.bError THEN
				bInsertAzure 	:= FALSE;
				nStateAzure 	:= 0;
				bErrorAzure 	:= FALSE;
				nErrorIDAzure 	:= fbMethodCall_DBRecordInsert.nErrorID;
			ELSE
				(* Error Occurred *)
				nStateAzure 	:= 6; 
				bErrorAzure	  	:= TRUE; 
				nErrorIDAzure 	:= fbMethodCall_DBRecordInsert.nErrorID;
			END_IF	
		END_IF
	
	6:
		;
END_CASE

ACTION M_Init:
(* Parameterize *)
SessionConnectInfo.tConnectTimeout 		:= T#1S;
SessionConnectInfo.tSessionTimeout 		:= T#1S;
SessionConnectInfo.sApplicationName		:= '';
// SessionConnectInfo.sApplicationUri 		:= '';
SessionConnectInfo.eSecurityMode 		:= eUASecurityMsgMode_None;
SessionConnectInfo.eSecurityPolicyUri 	:= eUASecurityPolicy_None;
SessionConnectInfo.eTransportProfileUri := eUATransportProfileUri_UATcp;
END_ACTION

END_PROGRAM

// ---- BECKHOFF SPECIFIC helper library/POUs/Database/UA_MethodCall_DBRecordInsert.TcPOU
FUNCTION_BLOCK UA_MethodCall_DBRecordInsert
VAR_INPUT
	bExecute			: BOOL;
	nConnectionHdl		: DWORD;
	nNamespaceIndex		: UINT; 			(* to be retrieved using UA_GetNamespaceIndex *)
	hDBID				: UDINT := 1; 
	pWriteData			: PVOID;
	cbWriteData			: UDINT;			(* Count of bytes to be read*)
	Timeout				: TIME := DEFAULT_ADS_TIMEOUT;
END_VAR
VAR_OUTPUT
	stUASQLState		: ST_UASQLState; 
	cbReadData_R		: UDINT; 
	bDone				: BOOL;
	bBusy				: BOOL;
	bError				: BOOL;
	nErrorID			: DWORD;
END_VAR
VAR
	iRdWrtReqState		: INT;
	RTrig				: R_TRIG;

	fbUA_MethodGetHandle: UA_MethodGetHandle;
	nMethodHdl			: DWORD;
	ObjectNodeID		: ST_UANodeID;
	MethodNodeID		: ST_UANodeID;

	fbUA_MethodCall		: UA_MethodCall;
	InputArguments		: ARRAY [1..nNumberOfInputArguments] OF ST_UAMethodArgInfo; (*ReadWriteReq has 6 input parameters *)
	nArg				: INT;
	nInputData			: ARRAY [1..nInputArgSize] OF BYTE; (* NetId(24) + Port(2)+ IG(4)+ IO(4) *)
	nOffset				: UDINT;
	stOutputArgInfo		: ARRAY [1..nNumberOfOutputArguments] OF ST_UAMethodArgInfo;
	{attribute 'hide'}
	nIndexOffset		: DINT := 16#1; 		(* IndexOffset*)
	
	fbUA_MethodReleaseHandle	: UA_MethodReleaseHandle;

	stDBRecordInsertRes	: ST_UAMethodCall_DBRecordInsertRes; 
	bInputDataError 	: BOOL;
END_VAR
VAR CONSTANT
	nInputArgSize			: UDINT := 34; (* NetId(24) + Port(2)+ IG(4)+ IO(4) *)
	nNumberOfInputArguments : UDINT := 6;
	nNumberOfOutputArguments : UDINT := 2;
	
	sNetID				: T_AmsNetId:='127.0.0.1.1.1'; 		(* AmsNetId OF the Target *)
	nPort				: INT := 21372;			(* Port number	*)	(* AMSPORT_DATABASESRV := 21372 = 16#537C*)
	nIndexGroup			: DINT := 16#80002;		(* IndexGroup*)		(* DBADS_IGR_DBRECORDINSERT *)
	cbReadData			: UDINT := SIZEOF(ST_UASQLState);			(* Count of bytes to be read*)
END_VAR

(*
ADSReadWriteReq(
******** Input Arguments ********
	string sNetID, 		: AmsNetId of the Target
	int16 Port,			: Port number	
	int32 IndexGroup,		: IndexGroup
	int32 IndexOffset,		: IndexOffset
	ByteString WriteData	: Data to be written to the device
	uint32 cbReadData		: Count of bytes to be read
******** Output Arguments ********
	bytestring Data		: count of bytes actually read
);
*)

RTrig(CLK:= bExecute);

CASE iRdWrtReqState OF

0:	(* Get Method Handle *)
	IF RTrig.Q THEN
		bBusy		:= TRUE;
		bDone 		:= FALSE;
		bError		:= FALSE;
		nErrorID	:= 0;
		ObjectNodeID.eIdentifierType := eUAIdentifierType_String;
		ObjectNodeID.nNamespaceIndex := nNamespaceIndex;
		ObjectNodeID.sIdentifier	 := 'ADSAMS';
	
		MethodNodeID.eIdentifierType := eUAIdentifierType_String;
		MethodNodeID.nNamespaceIndex := nNamespaceIndex;
		MethodNodeID.sIdentifier	 := 'ADSAMS.AdsReadWriteReq';

		M_Init();
		IF bInputDataError = FALSE THEN
			iRdWrtReqState 	:= iRdWrtReqState + 1;
		ELSE
			bBusy 		:= FALSE;
			bError 		:= TRUE;
			nErrorID 	:= DEVICE_INVALIDSIZE; //16#705 parameter size not correct
		END_IF
		MEMSET(ADR(stDBRecordInsertRes),0,SIZEOF(stDBRecordInsertRes));
		MEMSET(ADR(stUASQLState),0,SIZEOF(stUASQLState));
	END_IF


1:	(* Method Get Handle *)
	fbUA_MethodGetHandle(
			Execute			:= TRUE,
			ConnectionHdl	:= nConnectionHdl,
			ObjectNodeID	:= ObjectNodeID,
			MethodNodeID 	:= MethodNodeID,
			Timeout			:= Timeout,
			MethodHdl		=> nMethodHdl
		);
	IF NOT fbUA_MethodGetHandle.Busy THEN
		fbUA_MethodGetHandle(Execute := FALSE);

		IF NOT fbUA_MethodGetHandle.Error THEN
			(*  *)
			iRdWrtReqState := iRdWrtReqState + 1; (* Call Method *)
		ELSE
			bError			:= TRUE;
			nErrorID		:= fbUA_MethodGetHandle.ErrorID;
			iRdWrtReqState 	:= 3; (* Release Handle *)
		END_IF
	END_IF


2:	(* Method Call *)
	fbUA_MethodCall(
		Execute					:= TRUE,
		ConnectionHdl			:= nConnectionHdl,
		MethodHdl				:= nMethodHdl,
		nNumberOfInputArguments := nNumberOfInputArguments,		(* 6 *)
		pInputArgInfo			:= ADR(InputArguments),
		cbInputArgInfo			:= SIZEOF(InputArguments),
		pInputArgData			:= ADR(nInputData),
		cbInputArgData			:= nOffset,
		pInputWriteData			:= pWriteData,
		cbInputWriteData		:= cbWriteData,
		nNumberOfOutputArguments:= nNumberOfOutputArguments,		(* 2 *)
		pOutputArgInfo			:= ADR(stOutputArgInfo),
		cbOutputArgInfo			:= SIZEOF(stOutputArgInfo),
		pOutputArgInfoAndData	:= ADR(stDBRecordInsertRes),
		cbOutputArgInfoAndData	:= SIZEOF(stDBRecordInsertRes),
		Timeout					:= Timeout
	);
	IF NOT fbUA_MethodCall.Busy THEN
		fbUA_MethodCall(Execute := FALSE, cbRead_R => cbReadData_R);
		IF NOT fbUA_MethodCall.Error THEN
			(*  *)
			iRdWrtReqState 	:= iRdWrtReqState + 1; (* Release handle *)
			stUASQLState.nReturnCode := stDBRecordInsertRes.stSQLStateInternal.nReturnCode;
			(* ------------ copied from TcDatabase.lib *)
			IF stUASQLState.nReturnCode <> 0 THEN 
				bError := TRUE;
				nErrorID := stUASQLState.nReturnCode;
				stUASQLState.sSQLState		:= stDBRecordInsertRes.stSQLStateInternal.sSQLState;
				stUASQLState.nSQLErrorCode 	:= stDBRecordInsertRes.stSQLStateInternal.nSQLErrorCode;
			ELSE
				stUASQLState.sSQLState		:= '00000';	
				stUASQLState.nSQLErrorCode 	:= 0;		
			END_IF		
			(* ------------- copied from TcDatabase.lib *)
		ELSE
			bError			:= TRUE;
			nErrorID		:= fbUA_MethodCall.ErrorID;
			iRdWrtReqState	:= 3; (* Release handle *)
		END_IF
	END_IF


3:	(* Release Method Handle *)
	fbUA_MethodReleaseHandle(
		Execute			:= TRUE,
		ConnectionHdl	:= nConnectionHdl,
		MethodHdl		:= nMethodHdl,
		Timeout			:= Timeout
	);

	IF NOT fbUA_MethodReleaseHandle.Busy THEN
		fbUA_MethodReleaseHandle(Execute := FALSE);
		bBusy := FALSE;
		IF NOT fbUA_MethodReleaseHandle.Error THEN
			(* session closed *)
			bDone := TRUE;
			iRdWrtReqState 	:= 0; (* idle *)
		ELSE
			bError			:= TRUE;
			nErrorID		:= fbUA_MethodReleaseHandle.ErrorID;
			iRdWrtReqState 	:= 0; (* idle *)
		END_IF
	END_IF
END_CASE

ACTION M_Init:

//sNetID				:='127.0.0.1.1.1'; 		(* AmsNetId OF the Target *)
//nPort				:= 21372;					(* Port number	*)	(* AMSPORT_DATABASESRV := 21372 = 16#537C*)
//nIndexGroup			:= 16#80002;			(* IndexGroup*)		(* DBADS_IGR_DBRECORDINSERT *)
nIndexOffset		:= UDINT_TO_DINT(hDBID); 	(* IndexOffset*)
//cbReadData			:= SIZEOF(ST_UASQLState);	(* Count of bytes to be read*)

	
bInputDataError := FALSE; 
nOffset := 0;
MEMSET(ADR(InputArguments),0,SIZEOF(InputArguments));
MEMSET(ADR(nInputData),0,SIZEOF(nInputData));

nArg := 1;
(*sNetID := sAmsNetID;*)	(********** NET ID **********)
InputArguments[nArg].DataType			:= eUAType_String;
InputArguments[nArg].ValueRank			:= -1; 						(* Scalar = -1 or Array *)
InputArguments[nArg].ArrayDimensions[1]	:= 0; 						(* Number of Dimension in case its an array *)
InputArguments[nArg].nLenData			:= INT_TO_UDINT(LEN(sNetId)) + 1;	
IF nOffset + INT_TO_UDINT(LEN(sNetId))+1 > nInputArgSize THEN 
	bInputDataError := TRUE;
	RETURN;
ELSE
	MEMCPY(ADR(nInputData)+nOffset,ADR(sNetId),INT_TO_UDINT(LEN(sNetId))+1);			(* VALUE in BYTES FORM *)
	nOffset := nOffset + INT_TO_UDINT(LEN(sNetId))+1;
END_IF

nArg := nArg + 1;
(* nPort := 851;*)			(********** PORT **********)
InputArguments[nArg].DataType			:= eUAType_Int16;
InputArguments[nArg].ValueRank			:= -1; 						(* Scalar = -1 or Array *)
InputArguments[nArg].ArrayDimensions[1]	:= 0; 						(* Number of Dimension in case its an array *)
InputArguments[nArg].nLenData			:= SIZEOF(nPort);			(* Length if its a STRING *)
IF nOffset + SIZEOF(nPort) > nInputArgSize THEN 
	bInputDataError := TRUE;
	RETURN;
ELSE
	MEMCPY(ADR(nInputData)+nOffset,ADR(nPort),SIZEOF(nPort));			(* VALUE in BYTES FORM *)
	nOffset := nOffset + SIZEOF(nPort);
END_IF

nArg := nArg + 1;
(*nIndexGroup := 16#4020;*)	(********** INDEX GROUP **********)
InputArguments[nArg].DataType			:= eUAType_Int32;
InputArguments[nArg].ValueRank			:= -1; 							(* Scalar = -1 or Array *)
InputArguments[nArg].ArrayDimensions[1]	:= 0; 							(* Number of Dimension in case its an array *)
InputArguments[nArg].nLenData			:= SIZEOF(nIndexGroup);			(* Length if its a STRING *)
IF nOffset + SIZEOF(nIndexGroup) > nInputArgSize THEN 
	bInputDataError := TRUE;
	RETURN;
ELSE
	MEMCPY(ADR(nInputData)+nOffset,ADR(nIndexGroup),SIZEOF(nIndexGroup));		(* VALUE in BYTES FORM *)
	nOffset := nOffset + SIZEOF(nIndexGroup);
END_IF

nArg := nArg + 1;
(*nIndexOffset := 0; *)		(********** INDEX OFFSET **********)
InputArguments[nArg].DataType			:= eUAType_Int32;
InputArguments[nArg].ValueRank			:= -1; 							(* Scalar = -1 or Array *)
InputArguments[nArg].ArrayDimensions[1]	:= 0; 							(* Number of Dimension in case its an array *)
InputArguments[nArg].nLenData			:= SIZEOF(nIndexOffset);		(* Length if its a STRING *)
IF nOffset + SIZEOF(nIndexOffset) > nInputArgSize THEN 
	bInputDataError := TRUE;
	RETURN;
ELSE
	MEMCPY(ADR(nInputData)+nOffset,ADR(nIndexOffset),SIZEOF(nIndexOffset));	(* VALUE in BYTES FORM *)
	nOffset := nOffset + SIZEOF(nIndexOffset);
END_IF

nArg := nArg + 1;
(*Data := 2; *)		(*********** WriteData ***********)
InputArguments[nArg].DataType			:= eUAType_ByteString;
InputArguments[nArg].ValueRank			:= -1; 						(* Scalar = -1 or Array *)
InputArguments[nArg].ArrayDimensions[1]	:= 0; 						(* Number of Dimension in case its an array *)
InputArguments[nArg].nLenData			:= cbWriteData;				(* Length if its a STRING *)


nArg := nArg + 1;
(*Data := 2; *)		(*********** ReadData size ***********)
InputArguments[nArg].DataType			:= eUAType_UInt32;
InputArguments[nArg].ValueRank			:= -1; 						(* Scalar = -1 or Array *)
InputArguments[nArg].ArrayDimensions[1]	:= 0; 						(* Number of Dimension in case its an array *)
InputArguments[nArg].nLenData			:= SIZEOF(cbReadData);		(* Length if its a STRING *)


//************** Prepare Output Argument information ***********
stOutputArgInfo[1].nLenData := SIZEOF(stDBRecordInsertRes.stSQLStateInternal.nReturnCode);
stOutputArgInfo[2].nLenData := SIZEOF(stDBRecordInsertRes.stSQLStateInternal)- stOutputArgInfo[1].nLenData ;
END_ACTION

END_FUNCTION_BLOCK

// ---- Test_CloudSample/POUs/Helper/FB_BuildSQLInsert.TcPOU
FUNCTION_BLOCK FB_BuildSQLInsert
VAR_INPUT
	sTableName	:	STRING(12);
	stTimestamp	:	TIMESTRUCT;
	uiMesstellenID : UINT;
	stLogger	:	STRING(60);
	rMesswert	:	REAL;
	stEinheit	:	STRING(10);
	sValue		:	STRING(MAX_DATA_ACCURACY);
END_VAR
VAR_OUTPUT
	sQuery		:	STRING(100);
END_VAR
VAR
	sTemp		:	STRING(100);
	sTemp2		:	STRING(20);
	sYear 		:	STRING(4);
	sMonth		:	STRING(2);
	sDay		:	STRING(2);
	sHour		:	STRING(2);
	sMinute		:	STRING(2);
	sSecond		:	STRING(2);
	sMesswert	:	STRING(10);
	sMessId		:	STRING(5);
END_VAR

sYear := DWORD_TO_DECSTR(stTimestamp.wYear, 4);
sMonth := DWORD_TO_DECSTR(stTimestamp.wMonth, 2);
sDay := DWORD_TO_DECSTR(stTimestamp.wDay, 2);
sHour := DWORD_TO_DECSTR(stTimestamp.wHour, 2);
sMinute := DWORD_TO_DECSTR(stTimestamp.wMinute, 2);
sSecond := DWORD_TO_DECSTR(stTimestamp.wSecond, 2);
sMesswert := LREAL_TO_FMTSTR(rMesswert, 4, TRUE);
sMessId := DINT_TO_DECSTR(uiMesstellenID, 4);

sTemp2 := CONCAT(sYear, '-');
sTemp2 := CONCAT(sTemp2, sMonth);
sTemp2 := CONCAT(sTemp2, '-');
sTemp2 := CONCAT(sTemp2, sDay);
sTemp2 := CONCAT(sTemp2, ' ');
sTemp2 := CONCAT(sTemp2, sHour);
sTemp2 := CONCAT(sTemp2, ':');
sTemp2 := CONCAT(sTemp2, sMinute);
sTemp2 := CONCAT(sTemp2, ':');
sTemp2 := CONCAT(sTemp2, sSecond);

sTemp := CONCAT('INSERT INTO ', sTableName);
sTemp := CONCAT(sTemp, ' VALUES ($'');
sTemp := CONCAT(sTemp, sTemp2);
sTemp := CONCAT(sTemp, '$',');
sTemp := CONCAT(sTemp, sMessId);
sTemp := CONCAT(sTemp, ', $'');
sTemp := CONCAT(sTemp, stLogger);
sTemp := CONCAT(sTemp, '$', ');
sTemp := CONCAT(sTemp, sMesswert);
sTemp := CONCAT(sTemp, ', $'');
sTemp := CONCAT(sTemp, stEinheit);
sTemp := CONCAT(sTemp, '$')');

sQuery := sTemp;

END_FUNCTION_BLOCK

// ---- Test_Manz/POUs/PRG_CallTestMethodStringArray2Dim.TcPOU
PROGRAM PRG_CallTestMethodStringArray2Dim
VAR
	///CallInOutMultiParams(numberIn1(uInt32),numberIn2(UInt32),numberOut1(UInt32),numberOut2(UINT32));
	
	fbUA_Connect		: UA_Connect;
	SessionConnectInfo	: ST_UASessionConnectInfo;
	sOpcUA_URL			: STRING(MAX_STRING_LENGTH);
	nConnectionHdl		: DWORD;
	
	fbUA_GetNamespaceIndex	: UA_GetNamespaceIndex;
	nNamespaceIndex			: UINT;
	 
	fbUA_MethodGetHandle	: UA_MethodGetHandle;
	nMethodHdl				: DWORD;
	cbWriteData				: UDINT;
	ObjectNodeID			: ST_UANodeID;
	MethodNodeID			: ST_UANodeID;
	fbUA_MethodCall			: UA_MethodCall;
	InputArguments			: ARRAY[1..nNumberOfInputArguments] OF ST_UAMethodArgInfo;
	OutputArgInfo			: ARRAY [1..nNumberOfOutputArguments] OF ST_UAMethodArgInfo;
	nInputStringArray 		: ARRAY [1..3,1..3]  OF STRING;	
	nInputData				: ARRAY[1..nInputArgSize] OF BYTE;
	stOutputArgInfoAndData	: ST_UAMethodCall_CallTestMethodArray;
	
	fbUA_MethodReleaseHandle: UA_MethodReleaseHandle;
	
	fbUA_Disconnect	: UA_Disconnect;
	
	nArg			: INT;
	nOffset			: UDINT;
	bInputDataError	: BOOL;
	bTest			: BOOL := TRUE;
	bDone			: BOOL;
	bBusy			: BOOL;
	bError			: BOOL;
	nErrorID		: DWORD;
	iState			: INT;
END_VAR
VAR CONSTANT
	nNumberOfInputArguments : UDINT := 1;
	nNumberOfOutputArguments: UDINT := 2; 
	nInputArgSize 			: UDINT := 729;
END_VAR

(*
CallInOut1DimParams(	[numberIn1(uInt32),	numberIn2(UInt32)]
						[numberOut1(UInt32),numberOut2(UINT32),	numberOut3(UINT32)]
);
*)

CASE iState OF

0:	(* idle *)
	IF bTest THEN
		bTest		:= FALSE;
		bError		:= FALSE;
		nErrorID	:= 0;
		(* Parameterize *)
		sOpcUA_URL		:= 'opc.tcp://localhost:48032';	(* OpcUA Url of the device with ip address *)

		SessionConnectInfo.tConnectTimeout 		:= T#9M;
		SessionConnectInfo.tSessionTimeout 		:= T#9M;
		SessionConnectInfo.sApplicationName		:= '';
//		SessionConnectInfo.sApplicationUri 		:= '';
		SessionConnectInfo.eSecurityMode 		:= eUASecurityMsgMode_None;
		SessionConnectInfo.eSecurityPolicyUri 	:= eUASecurityPolicy_None;
		SessionConnectInfo.eTransportProfileUri := eUATransportProfileUri_UATcp;

		iState	:= iState + 1;
	END_IF

1:	(* open UA session *)
	fbUA_Connect(
		Execute				:= TRUE,
		ServerURL			:= sOpcUA_URL,
		SessionConnectInfo	:= SessionConnectInfo,
		Timeout				:= T#10S,
		ConnectionHdl		=> nConnectionHdl
	);

	IF NOT fbUA_Connect.Busy THEN
		fbUA_Connect(Execute := FALSE);

		IF NOT fbUA_Connect.Error THEN
			(* connected *)
			iState := iState + 1;
		ELSE
			bError			:= TRUE;
			nErrorID		:= fbUA_Connect.ErrorID;
			nConnectionHdl	:= 0;
			iState 			:= 0; (* idle *)
		END_IF
	END_IF


2:	(* GetNS Index *)
	fbUA_GetNamespaceIndex(
		Execute			:= TRUE,
		ConnectionHdl	:= nConnectionHdl,
		NamespaceUri	:= 'http://manz.com/ManzAddonTestForControl/',
		NamespaceIndex	=> nNamespaceIndex
	);

	IF NOT fbUA_GetNamespaceIndex.Busy THEN
		fbUA_GetNamespaceIndex(Execute := FALSE);

		IF NOT fbUA_GetNamespaceIndex.Error THEN
			(* namespace index read successfully *)
			iState 		:= iState + 1; (* get node handle *)
		ELSE
			bError		:= TRUE;
			nErrorID	:= fbUA_GetNamespaceIndex.ErrorID;
			iState 		:= 7; (* disconnect *)
		END_IF
	END_IF

3:	(* Get Method Handle *)
		ObjectNodeID.eIdentifierType := eUAIdentifierType_String;
		ObjectNodeID.nNamespaceIndex := nNamespaceIndex;
		ObjectNodeID.sIdentifier	:= 'ControlTest';
	
		MethodNodeID.eIdentifierType := eUAIdentifierType_String;
		MethodNodeID.nNamespaceIndex := nNamespaceIndex;
		MethodNodeID.sIdentifier	:= 'ControlTest.TestMethodArray';

		M_Init();
		IF bInputDataError = FALSE THEN
			iState 	:= iState + 1;
		ELSE
			bBusy		:= FALSE; 
			bError 		:= TRUE;
			nErrorID 	:= 16#70A; //out of memory
		END_IF


4:	(* Method Get Handle *)
	fbUA_MethodGetHandle(
			Execute			:= TRUE,
			ConnectionHdl	:= nConnectionHdl,
			ObjectNodeID	:= ObjectNodeID,
			MethodNodeID 	:= MethodNodeID,
			MethodHdl		=> nMethodHdl
		);
	IF NOT fbUA_MethodGetHandle.Busy THEN
		fbUA_MethodGetHandle(Execute := FALSE);

		IF NOT fbUA_MethodGetHandle.Error THEN
			(*  *)
			iState := iState + 1; (* Call Method *)
		ELSE
			bError		:= TRUE;
			nErrorID	:= fbUA_MethodGetHandle.ErrorID;
			iState	 	:= 6; (* Release method Handle *)
		END_IF
	END_IF


5:	(* Method Call *)

	fbUA_MethodCall(
		Execute					:= TRUE,
		Timeout					:= T#20S,
		ConnectionHdl			:= nConnectionHdl,
		MethodHdl				:= nMethodHdl,
		nNumberOfInputArguments := nNumberOfInputArguments,		(* 6 *)
		pInputArgData			:= ADR(nInputData),
		cbInputArgData			:= cbWriteData,
		pInputArgInfo			:= ADR(InputArguments),
		cbInputArgInfo			:= SIZEOF(InputArguments),
		nNumberOfOutputArguments:= nNumberOfOutputArguments,
		pOutputArgInfo			:= ADR(OutputArgInfo),
		cbOutputArgInfo			:= SIZEOF(OutputArgInfo),
		pOutputArgInfoAndData	:= ADR(stOutputArgInfoAndData),
		cbOutputArgInfoAndData	:= SIZEOF(stOutputArgInfoAndData)
	);
	IF NOT fbUA_MethodCall.Busy THEN
		fbUA_MethodCall(Execute := FALSE);

		IF NOT fbUA_MethodCall.Error THEN
			(*  *)
			iState 	:= iState + 1; (* Release handle *)
		ELSE
			bError		:= TRUE;
			nErrorID	:= fbUA_MethodCall.ErrorID;
			iState		:= 6; (* Release method handle *)
		END_IF
	END_IF


6:	(* Release Method Handle *)
	fbUA_MethodReleaseHandle(
		Execute			:= TRUE,
		ConnectionHdl	:= nConnectionHdl,
		MethodHdl		:= nMethodHdl
	);

	IF NOT fbUA_MethodReleaseHandle.Busy THEN
		fbUA_MethodReleaseHandle(Execute := FALSE);
		bBusy := FALSE;
		IF NOT fbUA_MethodReleaseHandle.Error THEN
			(* session closed *)
			iState 	:= 7; (* Disconnect *)
		ELSE
			bError		:= TRUE;
			nErrorID	:= fbUA_MethodReleaseHandle.ErrorID;
			iState 		:= 7; (* Disconnect *)
		END_IF
	END_IF
	
7:	(* Disconnect *) 
	fbUA_Disconnect(
		Execute			:= TRUE,
		ConnectionHdl	:= nConnectionHdl
	);

	IF NOT fbUA_Disconnect.Busy THEN
		fbUA_Disconnect(Execute := FALSE);

		IF NOT fbUA_Disconnect.Error THEN
			(* disconnected *)
			iState 			:= 0; (* idle *)
			bDone 	:= TRUE;
			bBusy 	:= FALSE;
		ELSE
			bBusy 	:= FALSE;
			bError			:= TRUE;
			nErrorID		:= fbUA_Disconnect.ErrorID;
			iState 			:= 0; (* idle *)
			nConnectionHdl	:= 0;
		END_IF
	END_IF
END_CASE

ACTION M_Init:
bInputDataError := FALSE; 
nOffset := 0;
MEMSET(ADR(InputArguments),0,SIZEOF(InputArguments));
MEMSET(ADR(nInputData),0,SIZEOF(nInputData));

nArg := 1;
(*numberIn1*)			(********** Input parameter 1 **********)
InputArguments[nArg].DataType			:= eUAType_String;
InputArguments[nArg].ValueRank			:= 2; 							(* Scalar = -1 or 1Dim-Array =1*)
InputArguments[nArg].ArrayDimensions[1]	:= 3; 							(* Number of Dimension in case its an array *)
InputArguments[nArg].ArrayDimensions[2]	:= 3; 		
InputArguments[nArg].nLenData			:= SIZEOF(nInputStringArray);			(* Length if its a STRING *)

IF nOffset + SIZEOF(nInputStringArray) > nInputArgSize THEN 
	bInputDataError := TRUE;
	RETURN;
ELSE
	MEMCPY(ADR(nInputData)+nOffset,ADR(nInputStringArray),SIZEOF(nInputStringArray));				(* VALUE in BYTES FORM *)
	nOffset := nOffset + SIZEOF(nInputStringArray);
END_IF

cbWriteData := nOffset;

//************** Prepare Output Argument information ***********
OutputArgInfo[1].nLenData := SIZEOF(stOutputArgInfoAndData.output1);
OutputArgInfo[2].nLenData := SIZEOF(stOutputArgInfoAndData.output2);
END_ACTION

END_PROGRAM

// ---- Test_Manz/POUs/PRG_CallTestMethodIntArray3Dim.TcPOU
PROGRAM PRG_CallTestMethodIntArray3Dim
VAR
	fbUA_Connect			: UA_Connect;
	SessionConnectInfo		: ST_UASessionConnectInfo;
	sOpcUA_URL				: STRING(MAX_STRING_LENGTH);
	nConnectionHdl			: DWORD;
	fbUA_GetNamespaceIndex	: UA_GetNamespaceIndex;
	nNamespaceIndex			: UINT;
	
	fbUA_MethodGetHandle	: UA_MethodGetHandle;
	nMethodHdl				: DWORD;
	ObjectNodeID			: ST_UANodeID;
	MethodNodeID			: ST_UANodeID;
	fbUA_MethodCall			: UA_MethodCall;
	InputArguments			: ARRAY[1..nNumberOfInputArguments] OF ST_UAMethodArgInfo;
	stOutputArgInfo			: ARRAY [1..nNumberOfOutputArguments] OF ST_UAMethodArgInfo;
	/// Bytes to be read 
	nInputData				: ARRAY[1..nInputArgSize] OF BYTE;
	/// Count of bytes to be written 
	cbWriteData: UDINT;
	///CallInOutMultiParams(numberIn1(uInt32),numberIn2(UInt32),numberOut1(UInt32),numberOut2(UINT32));
	//numberIn3Dim: ARRAY[1..3,1..3,1..3] OF UDINT := [1,2,3,4,5,6,7,8,9,10,11,12,13,14,15,16,17,18,19,20,21,22,23,24,25,26,27];
	numberIn3Dim			: ARRAY[1..2,1..2,1..2] OF DINT := [1,2,3,4,5,6,7,8];
	OutputArgAndData		: ST_UAMethodCall_CallTestMethodIntArray3Dim;
	
	fbUA_MethodReleaseHandle	: UA_MethodReleaseHandle;
	
	fbUA_Disconnect	: UA_Disconnect;
	
	bTest			: BOOL := TRUE;
	bDone			: BOOL;
	bBusy			: BOOL;
	bError			: BOOL;
	nErrorID		: DWORD;
	iState			: INT;
	nOffset			: UDINT;
	nArg			: INT;
	bInputDataError	: BOOL;
END_VAR
VAR CONSTANT
	nNumberOfInputArguments : UDINT := 1;
	nNumberOfOutputArguments: UDINT := 1; 
	nInputArgSize 			: UDINT := 32;
END_VAR

(*
CallInOut1DimParams(	[numberIn1(uInt32),	numberIn2(UInt32)]
						[numberOut1(UInt32),numberOut2(UINT32),	numberOut3(UINT32)]
);
*)

CASE iState OF

0:	(* idle *)
	IF bTest THEN
		bTest		:= FALSE;
		bError		:= FALSE;
		nErrorID	:= 0;
		(* Parameterize *)
		//sOpcUA_URL		:= 'opc.tcp://localhost:48032';	(* OpcUA Url of the device with ip address *)
		sOpcUA_URL		:= 'opc.tcp://localhost-nb:4842';	(* OpcUA Url of the device with ip address *)

		SessionConnectInfo.tConnectTimeout 		:= T#9M;
		SessionConnectInfo.tSessionTimeout 		:= T#9M;
		SessionConnectInfo.sApplicationName		:= '';
//		SessionConnectInfo.sApplicationUri 		:= '';
		SessionConnectInfo.eSecurityMode 		:= eUASecurityMsgMode_None;
		SessionConnectInfo.eSecurityPolicyUri 	:= eUASecurityPolicy_None;
		SessionConnectInfo.eTransportProfileUri := eUATransportProfileUri_UATcp;

		iState	:= iState + 1;
	END_IF


1:	(* open UA session *)
	fbUA_Connect(
		Execute				:= TRUE,
		ServerURL			:= sOpcUA_URL,
		SessionConnectInfo	:= SessionConnectInfo,
		Timeout				:= T#10S,
		ConnectionHdl		=> nConnectionHdl
	);

	IF NOT fbUA_Connect.Busy THEN
		fbUA_Connect(Execute := FALSE);

		IF NOT fbUA_Connect.Error THEN
			(* connected *)
			iState := iState + 1;
		ELSE
			bError			:= TRUE;
			nErrorID		:= fbUA_Connect.ErrorID;
			nConnectionHdl	:= 0;
			iState 			:= 0; (* idle *)
		END_IF
	END_IF


2:	(* GetNS Index *)
	fbUA_GetNamespaceIndex(
		Execute			:= TRUE,
		ConnectionHdl	:= nConnectionHdl,
		NamespaceUri	:= 'http://manz.com/ManzAddonTestForControl/',
		NamespaceIndex	=> nNamespaceIndex
	);

	IF NOT fbUA_GetNamespaceIndex.Busy THEN
		fbUA_GetNamespaceIndex(Execute := FALSE);

		IF NOT fbUA_GetNamespaceIndex.Error THEN
			(* namespace index read successfully *)
			iState 		:= iState + 1; (* get node handle *)
		ELSE
			bError		:= TRUE;
			nErrorID	:= fbUA_GetNamespaceIndex.ErrorID;
			iState 		:= 7; (* disconnect *)
		END_IF
	END_IF

3:	(* Get Method Handle *)
		ObjectNodeID.eIdentifierType := eUAIdentifierType_String;
		ObjectNodeID.nNamespaceIndex := nNamespaceIndex;
		ObjectNodeID.sIdentifier	:= 'ControlTest';
	
		MethodNodeID.eIdentifierType := eUAIdentifierType_String;
		MethodNodeID.nNamespaceIndex := nNamespaceIndex;
		MethodNodeID.sIdentifier	:= 'ControlTest.TestMethodIntArray3Dim';

		M_Init();
		IF bInputDataError = FALSE THEN
			iState 	:= iState + 1;
		ELSE
			bBusy		:= FALSE; 
			bError 		:= TRUE;
			nErrorID 	:= 16#70A; //out of memory
		END_IF


4:	(* Method Get Handle *)
	fbUA_MethodGetHandle(
			Execute			:= TRUE,
			ConnectionHdl	:= nConnectionHdl,
			ObjectNodeID	:= ObjectNodeID,
			MethodNodeID 	:= MethodNodeID,
			MethodHdl		=> nMethodHdl
		);
	IF NOT fbUA_MethodGetHandle.Busy THEN
		fbUA_MethodGetHandle(Execute := FALSE);

		IF NOT fbUA_MethodGetHandle.Error THEN
			(*  *)
			iState := iState + 1; (* Call Method *)
		ELSE
			bError		:= TRUE;
			nErrorID	:= fbUA_MethodGetHandle.ErrorID;
			iState	 	:= 6; (* Release method Handle *)
		END_IF
	END_IF


5:	(* Method Call *)
	fbUA_MethodCall(
		Execute					:= TRUE,
		Timeout					:= T#20S,
		ConnectionHdl			:= nConnectionHdl,
		MethodHdl				:= nMethodHdl,
		nNumberOfInputArguments := nNumberOfInputArguments,		(* 1 *)
		pInputArgData			:= ADR(nInputData),
		cbInputArgData			:= cbWriteData,
		pInputArgInfo			:= ADR(InputArguments),
		cbInputArgInfo			:= SIZEOF(InputArguments),
		nNumberOfOutputArguments:= nNumberOfOutputArguments,
		pOutputArgInfo			:= ADR(stOutputArgInfo),
		cbOutputArgInfo			:= SIZEOF(stOutputArgInfo),
		pOutputArgInfoAndData	:= ADR(OutputArgAndData),
		cbOutputArgInfoAndData	:= SIZEOF(OutputArgAndData),
			
	);
	IF NOT fbUA_MethodCall.Busy THEN
		fbUA_MethodCall(Execute := FALSE);

		IF NOT fbUA_MethodCall.Error THEN
			(*  *)
			iState 	:= iState + 1; (* Release handle *)
		ELSE
			bError		:= TRUE;
			nErrorID	:= fbUA_MethodCall.ErrorID;
			iState		:= 6; (* Release method handle *)
		END_IF
	END_IF


6:	(* Release Method Handle *)
	fbUA_MethodReleaseHandle(
		Execute			:= TRUE,
		ConnectionHdl	:= nConnectionHdl,
		MethodHdl		:= nMethodHdl
	);

	IF NOT fbUA_MethodReleaseHandle.Busy THEN
		fbUA_MethodReleaseHandle(Execute := FALSE);
		bBusy := FALSE;
		IF NOT fbUA_MethodReleaseHandle.Error THEN
			(* session closed *)
			iState 	:= 7; (* Disconnect *)
		ELSE
			bError		:= TRUE;
			nErrorID	:= fbUA_MethodReleaseHandle.ErrorID;
			iState 		:= 7; (* Disconnect *)
		END_IF
	END_IF
	
7:	(* Disconnect *) 
	fbUA_Disconnect(
		Execute			:= TRUE,
		ConnectionHdl	:= nConnectionHdl
	);

	IF NOT fbUA_Disconnect.Busy THEN
		fbUA_Disconnect(Execute := FALSE);

		IF NOT fbUA_Disconnect.Error THEN
			(* disconnected *)
			iState 			:= 0; (* idle *)
			bDone 	:= TRUE;
			bBusy 	:= FALSE;
		ELSE
			bBusy 	:= FALSE;
			bError			:= TRUE;
			nErrorID		:= fbUA_Disconnect.ErrorID;
			iState 			:= 0; (* idle *)
			nConnectionHdl	:= 0;
		END_IF
	END_IF
END_CASE

ACTION M_Init:
bInputDataError := FALSE; 
nOffset := 0;
MEMSET(ADR(InputArguments),0,SIZEOF(InputArguments));
MEMSET(ADR(nInputData),0,SIZEOF(nInputData));

nArg := 1;
(*numberIn1*)			(********** Input parameter 1 **********)
InputArguments[nArg].DataType			:= eUAType_Int32;
InputArguments[nArg].ValueRank			:= 3; 							(* Scalar = -1 or 1Dim-Array =1*)
InputArguments[nArg].ArrayDimensions[1]	:= 2; 							(* Number of Dimension in case its an array *)
InputArguments[nArg].ArrayDimensions[2]	:= 2; 
InputArguments[nArg].ArrayDimensions[3]	:= 2; 		
InputArguments[nArg].nLenData			:= SIZEOF(numberIn3Dim);			(* Length if its a STRING *)

IF nOffset + SIZEOF(numberIn3Dim) > nInputArgSize THEN 
	bInputDataError := TRUE;
	RETURN;
ELSE
	MEMCPY(ADR(nInputData)+nOffset,ADR(numberIn3Dim),SIZEOF(numberIn3Dim));				(* VALUE in BYTES FORM *)
	nOffset := nOffset + SIZEOF(numberIn3Dim);
END_IF

cbWriteData := nOffset;

//************** Prepare Output Argument information ***********
stOutputArgInfo[1].nLenData := SIZEOF(OutputArgAndData.output1);
END_ACTION

END_PROGRAM

// ---- Tests_Henning/POUs/PRG_2DArrayTest.TcPOU
PROGRAM PRG_2DArrayTest
VAR
	iState: INT := 3; //we need to wait for UAServer to provide variables
END_VAR

CASE iState OF
0:	
	PRG_2DArrayTest_Read();
	IF(NOT PRG_2DArrayTest_Read.bBusy AND NOT PRG_2DArrayTest_Read.bError) THEN
		iState := iState+1;
	END_IF
1:
	PRG_2DArrayTest_Write();
	IF(NOT PRG_2DArrayTest_Write.bBusy AND NOT PRG_2DArrayTest_Write.bError) THEN
		iState := iState+1;
	END_IF
2:
	PRG_2DArrayTest_ReadWritten();
	IF(NOT PRG_2DArrayTest_ReadWritten.bBusy AND NOT PRG_2DArrayTest_ReadWritten.bError) THEN
		iState := iState+1;
	END_IF
END_CASE

END_PROGRAM

// ---- Tests_Henning/POUs/PRG_2DArrayTest_Read.TcPOU
PROGRAM PRG_2DArrayTest_Read
VAR
	fbUA_Connect: UA_Connect;
	SessionConnectInfo: ST_UASessionConnectInfo;
	nConnectionHdl: DWORD;
	fbUA_GetNamespaceIndex: UA_GetNamespaceIndex;
	nNamespaceIndex: UINT;
	fbUA_NodeGetHandle: UA_NodeGetHandle;
	NodeID: ST_UANodeID;
	nNodeHdl: DWORD;
	fbUA_Read: UA_Read;
	stIndexRange: ARRAY[1..nMaxIndexRange] OF ST_UAIndexRange;
	nIndexRangeCount: UINT;
	stNodeAddInfo: ST_UANodeAdditionalInfo;
	Variable: ARRAY[1..nMaxReadData] OF BYTE;
	///DINT; 		// change the data type according to the variable type to be read
	nReadData: STRING;
	fbUA_NodeReleaseHandle: UA_NodeReleaseHandle;
	fbUA_Disconnect: UA_Disconnect;
	iState: INT;
	bTest: BOOL := TRUE;
	bDone: BOOL;
	bBusy: BOOL;
	bError: BOOL;
	nErrorID: DWORD;
	nLoopVars: UINT;
END_VAR

CASE iState OF
0:	(* idle *)
	IF bTest THEN
		bTest		:= FALSE;
		bError		:= FALSE;
		nErrorID	:= 0;
		bBusy 		:= TRUE; 
		SessionConnectInfo.tConnectTimeout 		:= T#9S;
		SessionConnectInfo.tSessionTimeout 		:= T#9S;
		SessionConnectInfo.sApplicationName		:= '';
		SessionConnectInfo.sApplicationUri 		:= '';
		SessionConnectInfo.eSecurityMode 		:= eUASecurityMsgMode_None;
		SessionConnectInfo.eSecurityPolicyUri 	:= eUASecurityPolicy_None;
		SessionConnectInfo.eTransportProfileUri := eUATransportProfileUri_UATcp;

		stNodeAddInfo.nIndexRangeCount := nIndexRangeCount;
		stNodeAddInfo.stIndexRange := stIndexRange;
		iState	:= iState + 1;
	END_IF

1:	(* open UA session *)
	fbUA_Connect(
		Execute				:= TRUE,
		ServerURL			:= GVL_ArrayTests2DimPLC.sOpcUA_URL,
		SessionConnectInfo	:= SessionConnectInfo,
		Timeout				:= T#10S,
		ConnectionHdl		=> nConnectionHdl
	);

	IF NOT fbUA_Connect.Busy THEN
		fbUA_Connect(Execute := FALSE);

		IF NOT fbUA_Connect.Error THEN
			(* session open *)
			iState := iState + 1;
		ELSE
			bError			:= TRUE;
			nErrorID		:= fbUA_Connect.ErrorID;
			nConnectionHdl	:= 0;
			iState 			:= 0; (* idle *)
		END_IF
	END_IF


2:	(* GetNS Index *)
	IF NOT GVL_ArrayTests2DimPLC.NodeID_DoOrDont[nLoopVars] THEN
		iState := 6;
	END_IF
	fbUA_GetNamespaceIndex(
		Execute			:= TRUE,
		ConnectionHdl	:= nConnectionHdl,
		NamespaceUri	:= GVL_ArrayTests2DimPLC.sNodeIDNamespace,
		NamespaceIndex	=> nNamespaceIndex
	);

	IF NOT fbUA_GetNamespaceIndex.Busy THEN
		fbUA_GetNamespaceIndex(Execute := FALSE);

		IF NOT fbUA_GetNamespaceIndex.Error THEN
			(* session closed *)
			iState 		:= iState + 1; (* idle *)
		ELSE
			bError		:= TRUE;
			nErrorID	:= fbUA_GetNamespaceIndex.ErrorID;
			iState 		:= 6; (* idle *)
		END_IF
	END_IF


3:	(* Get Node Handle *)
	NodeID.eIdentifierType := eUAIdentifierType_String;
	NodeID.nNamespaceIndex := nNamespaceIndex;
	NodeID.sIdentifier	:= GVL_ArrayTests2DimPLC.NodeID_Identifiers[nLoopVars]; // 'GVL_static.stat_BSTR_0';
	fbUA_NodeGetHandle(
		Execute			:= TRUE,
		ConnectionHdl	:= nConnectionHdl,
		NodeID			:= NodeID,
		NodeHdl			=> nNodeHdl
	);

	IF NOT fbUA_NodeGetHandle.Busy THEN
		fbUA_NodeGetHandle(Execute := FALSE);

		IF NOT fbUA_NodeGetHandle.Error THEN
			(* session closed *)
			iState 		:= iState + 1; (* idle *)
		ELSE
			bError		:= TRUE;
			nErrorID	:= fbUA_NodeGetHandle.ErrorID;
			iState 		:= 6; (* idle *)
		END_IF
	END_IF


4: 	(* UA_Read *)
	fbUA_Read(
		Execute			:= TRUE,
		ConnectionHdl	:= nConnectionHdl,
		NodeHdl			:= nNodeHdl,
		stNodeAddInfo 	:= stNodeAddInfo,
		cbData			:= GVL_ArrayTests2DimPLC.NodeID_Sizes[nLoopVars], //SIZEOF(nReadData),
		pVariable		:= ADR(GVL_ArrayTests2DimPLC.NodeID_ReadResults[nLoopVars].nData) //Variable
		);

	IF NOT fbUA_Read.Busy THEN
		fbUA_Read(
			Execute 	:= FALSE);

		IF NOT fbUA_Read.Error THEN
			(* session closed *)
			iState 		:= iState + 1; (* idle *)
			//Do we need this? We simply store in UNION! MEMCPY(ADR(nReadData),ADR(Variable),SIZEOF(nReadData));
		ELSE
			bError		:= TRUE;
			nErrorID	:= fbUA_Read.ErrorID;
			iState 		:= 7; (* idle *)
		END_IF
	END_IF



5:	(* Release Node Handle *)
	fbUA_NodeReleaseHandle(
		Execute			:= TRUE,
		ConnectionHdl	:= nConnectionHdl,
		NodeHdl			:= nNodeHdl
	);

	IF NOT fbUA_NodeReleaseHandle.Busy THEN
		fbUA_NodeReleaseHandle(Execute := FALSE);

		IF NOT fbUA_NodeReleaseHandle.Error THEN
			(* session closed *)
			iState 		:= iState + 1; (* idle *)
		ELSE
			bError		:= TRUE;
			nErrorID	:= fbUA_NodeReleaseHandle.ErrorID;
			iState 		:= 6; (* idle *)
		END_IF
	END_IF


6:	(* close session *)
	fbUA_Disconnect(
		Execute			:= TRUE,
		ConnectionHdl	:= nConnectionHdl
	);

	IF NOT fbUA_Disconnect.Busy THEN
		fbUA_Disconnect(Execute := FALSE);

		IF NOT fbUA_Disconnect.Error THEN
			(* session closed *)
			iState 		:= 0; (* idle *)
			//restart with next var, if existing in array
			IF(nLoopVars < nEndOfNodeIDVarsArray_2Dim) THEN
				nLoopVars := nLoopVars+1;
				bTest := TRUE;
			ELSE 
				bBusy 		:= FALSE;
				//prepare for next call 
				bTest := TRUE;
				nLoopVars := 0;
			END_IF
		ELSE
			bError			:= TRUE;
			nErrorID		:= fbUA_Disconnect.ErrorID;
			iState 			:= 0; (* idle *)
			nConnectionHdl	:= 0;
		END_IF
	END_IF
END_CASE

END_PROGRAM

// ---- Tests_Henning/POUs/PRG_2DArrayTest_Write.TcPOU
PROGRAM PRG_2DArrayTest_Write
VAR
	fbUA_Connect: UA_Connect;
	SessionConnectInfo: ST_UASessionConnectInfo;
	sOpcUA_URL: STRING(MAX_STRING_LENGTH);
	nConnectionHdl: DWORD;
	fbUA_GetNamespaceIndex: UA_GetNamespaceIndex;
	sNamespaceUri: STRING(MAX_STRING_LENGTH);
	nNamespaceIndex: UINT;
	fbUA_NodeGetHandle: UA_NodeGetHandle;
	NodeID: ST_UANodeID;
	nNodeHdl: DWORD;
	fbUA_Write: UA_Write;
	stIndexRange: ARRAY[1..nMaxIndexRange] OF ST_UAIndexRange;
	nIndexRangeCount: UINT;
	stNodeAddInfo: ST_UANodeAdditionalInfo;
	/// UDINT := 12312345;		// change according to the type of variable
	nWriteData: STRING := 'Hallo';
	Variable: ARRAY[1..nMaxReadData] OF BYTE;
	cbData: UDINT;
	fbUA_NodeReleaseHandle: UA_NodeReleaseHandle;
	fbUA_Disconnect: UA_Disconnect;
	iState: INT;
	bTest: BOOL := TRUE;
	bDone: BOOL;
	bBusy: BOOL;
	bError: BOOL;
	nErrorID: DWORD;
	nLoopVars: UINT;
END_VAR

CASE iState OF
0:	(* idle *)
	IF bTest THEN
		bTest	:= FALSE;
		bError	:= FALSE;
		nErrorID	:= 0;
		bBusy := TRUE; 

		(* Parameterize 
		GVL_ScalarTests.NodeID_WriteCommands[0].bBool := TRUE; 
		GVL_ScalarTests.NodeID_WriteCommands[1].sString := 'WriteTest'; 
		GVL_ScalarTests.NodeID_WriteCommands[2].bByte := 123; 
		GVL_ScalarTests.NodeID_WriteCommands[3].nInt := 124; 
		GVL_ScalarTests.NodeID_WriteCommands[4].nUdint := 125; 
		GVL_ScalarTests.NodeID_WriteCommands[5].nLReal := 1.23456; //R8x 
		GVL_ScalarTests.NodeID_WriteCommands[6].bByte := 111; 
		GVL_ScalarTests.NodeID_WriteCommands[7].nInt := 112; 
		GVL_ScalarTests.NodeID_WriteCommands[8].nUdint := 113; 
		*)
		
		SessionConnectInfo.tConnectTimeout 		:= T#9S;
		SessionConnectInfo.tSessionTimeout 		:= T#9S;
		SessionConnectInfo.sApplicationName		:= '';
		SessionConnectInfo.sApplicationUri 		:= '';
		SessionConnectInfo.eSecurityMode 		:= eUASecurityMsgMode_None;
		SessionConnectInfo.eSecurityPolicyUri 	:= eUASecurityPolicy_None;
		SessionConnectInfo.eTransportProfileUri := eUATransportProfileUri_UATcp;
		
		stNodeAddInfo.nIndexRangeCount := nIndexRangeCount;
		stNodeAddInfo.stIndexRange := stIndexRange;
		iState	:= iState + 1;
	END_IF

1:	(* open UA session *)
	fbUA_Connect(
		Execute				:= TRUE,
		ServerURL			:= GVL_ArrayTests2DimPLC.sOpcUA_URL,
		SessionConnectInfo	:= SessionConnectInfo,
		Timeout				:= T#10S,
		ConnectionHdl		=> nConnectionHdl
	);

	IF NOT fbUA_Connect.Busy THEN
		fbUA_Connect(Execute := FALSE);

		IF NOT fbUA_Connect.Error THEN
			(* session open *)
			iState := iState + 1;
		ELSE
			bError			:= TRUE;
			nErrorID		:= fbUA_Connect.ErrorID;
			nConnectionHdl	:= 0;
			iState 			:= 0; (* idle *)
		END_IF
	END_IF


2:	(* GetNS Index *)
	IF NOT GVL_ArrayTests2DimPLC.NodeID_DoOrDont[nLoopVars] THEN
		iState := 6;
	END_IF
	fbUA_GetNamespaceIndex(
		Execute			:= TRUE,
		ConnectionHdl	:= nConnectionHdl,
		NamespaceUri	:= GVL_ArrayTests2DimPLC.sNodeIDNamespace,
		NamespaceIndex	=> nNamespaceIndex
	);

	IF NOT fbUA_GetNamespaceIndex.Busy THEN
		fbUA_GetNamespaceIndex(Execute := FALSE);

		IF NOT fbUA_GetNamespaceIndex.Error THEN
			(* session closed *)
			iState 		:= iState + 1; (* idle *)
		ELSE
			bError		:= TRUE;
			nErrorID	:= fbUA_GetNamespaceIndex.ErrorID;
			iState 		:= 6; (* idle *)
		END_IF
	END_IF


3:	(* Get Node Handle *)
	NodeID.eIdentifierType := eUAIdentifierType_String;
	NodeID.nNamespaceIndex := nNamespaceIndex;
	NodeID.sIdentifier	:= GVL_ArrayTests2DimPLC.NodeID_Identifiers[nLoopVars]; // 'GVL_static.stat_BSTR_0';
	fbUA_NodeGetHandle(
		Execute			:= TRUE,
		ConnectionHdl	:= nConnectionHdl,
		NodeID			:= NodeID,
		NodeHdl			=> nNodeHdl
	);

	IF NOT fbUA_NodeGetHandle.Busy THEN
		fbUA_NodeGetHandle(Execute := FALSE);

		IF NOT fbUA_NodeGetHandle.Error THEN
			(* session closed *)
			IF SIZEOF(nWriteData) <= nMaxReadData THEN 
				iState 		:= iState + 1; (* idle *)
				MEMSET(ADR(Variable),0,SIZEOF(Variable));
				MEMCPY(ADR(Variable),ADR(nWriteData),SIZEOF(nWriteData));
			ELSE
				//cannot write buffer too small -> increase the value of nMaxData in GVL
				bError		:= TRUE;
				iState 		:= 6; (* idle *)
			END_IF
		ELSE
			bError		:= TRUE;
			nErrorID	:= fbUA_NodeGetHandle.ErrorID;
			iState 		:= 6; (* idle *)
		END_IF
	END_IF


4: 	(* UA_Write *)
	fbUA_Write(
		Execute			:= TRUE,
		ConnectionHdl	:= nConnectionHdl,
		NodeHdl			:= nNodeHdl,
		stNodeAddInfo	:= stNodeAddInfo,
		cbData			:= GVL_ArrayTests2DimPLC.NodeID_Sizes[nLoopVars], //SIZEOF(nWriteData),
		pVariable		:= ADR(GVL_ArrayTests2DimPLC.NodeID_WriteCommands[nLoopVars].nData) // Variable		:= Variable
		);

	IF NOT fbUA_Write.Busy THEN
		fbUA_Write(
			Execute 		:= FALSE);

		IF NOT fbUA_Write.Error THEN
			(* session closed *)
			iState 		:= iState + 1; (* idle *)
		ELSE
			bError		:= TRUE;
			nErrorID	:= fbUA_Write.ErrorID;
			iState 		:= 7; (* idle *)
		END_IF
	END_IF


5:	(* Release Node Handle *)
	fbUA_NodeReleaseHandle(
		Execute			:= TRUE,
		ConnectionHdl	:= nConnectionHdl,
		NodeHdl			:= nNodeHdl
	);

	IF NOT fbUA_NodeReleaseHandle.Busy THEN
		fbUA_NodeReleaseHandle(Execute := FALSE);

		IF NOT fbUA_NodeReleaseHandle.Error THEN
			(* session closed *)
			iState 		:= iState + 1; (* idle *)
		ELSE
			bError		:= TRUE;
			nErrorID	:= fbUA_NodeReleaseHandle.ErrorID;
			iState 		:= 6; (* idle *)
		END_IF
	END_IF


6:	(* close session *)
	fbUA_Disconnect(
		Execute			:= TRUE,
		ConnectionHdl	:= nConnectionHdl
	);

	IF NOT fbUA_Disconnect.Busy THEN
		fbUA_Disconnect(Execute := FALSE);

		IF NOT fbUA_Disconnect.Error THEN
			(* session closed *)
			iState 		:= 0; (* idle *)			//restart with next var, if existing in array
			IF(nLoopVars < nEndOfNodeIDVarsArray_2Dim) THEN
				nLoopVars := nLoopVars+1;
				bTest := TRUE;
			ELSE 
				bBusy 		:= FALSE;
				//prepare for next call
				bTest := TRUE; 
				nLoopVars := 0;
			END_IF
		ELSE
			bError		:= TRUE;
			nErrorID	:= fbUA_Disconnect.ErrorID;
			iState 		:= 0; (* idle *)
			nConnectionHdl	:= 0;
		END_IF
	END_IF
END_CASE

END_PROGRAM

// ---- Tests_Henning/POUs/PRG_2DArrayTest_ReadWritten.TcPOU
PROGRAM PRG_2DArrayTest_ReadWritten
VAR
	fbUA_Connect: UA_Connect;
	SessionConnectInfo: ST_UASessionConnectInfo;
	nConnectionHdl: DWORD;
	fbUA_GetNamespaceIndex: UA_GetNamespaceIndex;
	nNamespaceIndex: UINT;
	fbUA_NodeGetHandle: UA_NodeGetHandle;
	NodeID: ST_UANodeID;
	nNodeHdl: DWORD;
	fbUA_Read: UA_Read;
	stIndexRange: ARRAY[1..nMaxIndexRange] OF ST_UAIndexRange;
	nIndexRangeCount: UINT;
	stNodeAddInfo: ST_UANodeAdditionalInfo;
	Variable: ARRAY[1..nMaxReadData] OF BYTE;
	///DINT; 		// change the data type according to the variable type to be read
	nReadData: STRING;
	fbUA_NodeReleaseHandle: UA_NodeReleaseHandle;
	fbUA_Disconnect: UA_Disconnect;
	iState: INT;
	bTest: BOOL := TRUE;
	bDone: BOOL;
	bBusy: BOOL;
	bError: BOOL;
	nErrorID: DWORD;
	nLoopVars: UINT;
	counter: UDINT;
	a: ARRAY[1..nMaxReadDataArray_2Dim] OF BYTE;
	b: ARRAY[1..nMaxReadDataArray_2Dim] OF BYTE;
	a_: BYTE;
	b_: BYTE;
	nTmpL: UINT;
END_VAR

CASE iState OF
0:	(* idle *)
	IF bTest THEN
		bTest		:= FALSE;
		bError		:= FALSE;
		nErrorID	:= 0;
		bBusy 		:= TRUE; 
		SessionConnectInfo.tConnectTimeout 		:= T#9S;
		SessionConnectInfo.tSessionTimeout 		:= T#9S;
		SessionConnectInfo.sApplicationName		:= '';
		SessionConnectInfo.sApplicationUri 		:= '';
		SessionConnectInfo.eSecurityMode 		:= eUASecurityMsgMode_None;
		SessionConnectInfo.eSecurityPolicyUri 	:= eUASecurityPolicy_None;
		SessionConnectInfo.eTransportProfileUri := eUATransportProfileUri_UATcp;

		stNodeAddInfo.nIndexRangeCount := nIndexRangeCount;
		stNodeAddInfo.stIndexRange := stIndexRange;
		iState	:= iState + 1;
	END_IF

1:	(* open UA session *)
	fbUA_Connect(
		Execute				:= TRUE,
		ServerURL			:= GVL_ArrayTests2DimPLC.sOpcUA_URL,
		SessionConnectInfo	:= SessionConnectInfo,
		Timeout				:= T#10S,
		ConnectionHdl		=> nConnectionHdl
	);

	IF NOT fbUA_Connect.Busy THEN
		fbUA_Connect(Execute := FALSE);

		IF NOT fbUA_Connect.Error THEN
			(* session open *)
			iState := iState + 1;
		ELSE
			bError			:= TRUE;
			nErrorID		:= fbUA_Connect.ErrorID;
			nConnectionHdl	:= 0;
			iState 			:= 0; (* idle *)
		END_IF
	END_IF


2:	(* GetNS Index *)
	IF NOT GVL_ArrayTests2DimPLC.NodeID_DoOrDont[nLoopVars] THEN
		iState := 6;
	END_IF
	fbUA_GetNamespaceIndex(
		Execute			:= TRUE,
		ConnectionHdl	:= nConnectionHdl,
		NamespaceUri	:= GVL_ArrayTests2DimPLC.sNodeIDNamespace,
		NamespaceIndex	=> nNamespaceIndex
	);

	IF NOT fbUA_GetNamespaceIndex.Busy THEN
		fbUA_GetNamespaceIndex(Execute := FALSE);

		IF NOT fbUA_GetNamespaceIndex.Error THEN
			(* session closed *)
			iState 		:= iState + 1; (* idle *)
		ELSE
			bError		:= TRUE;
			nErrorID	:= fbUA_GetNamespaceIndex.ErrorID;
			iState 		:= 6; (* idle *)
		END_IF
	END_IF


3:	(* Get Node Handle *)
	NodeID.eIdentifierType := eUAIdentifierType_String;
	NodeID.nNamespaceIndex := nNamespaceIndex;
	NodeID.sIdentifier	:= GVL_ArrayTests2DimPLC.NodeID_Identifiers[nLoopVars]; // 'GVL_static.stat_BSTR_0';
	fbUA_NodeGetHandle(
		Execute			:= TRUE,
		ConnectionHdl	:= nConnectionHdl,
		NodeID			:= NodeID,
		NodeHdl			=> nNodeHdl
	);

	IF NOT fbUA_NodeGetHandle.Busy THEN
		fbUA_NodeGetHandle(Execute := FALSE);

		IF NOT fbUA_NodeGetHandle.Error THEN
			(* session closed *)
			iState 		:= iState + 1; (* idle *)
		ELSE
			bError		:= TRUE;
			nErrorID	:= fbUA_NodeGetHandle.ErrorID;
			iState 		:= 6; (* idle *)
		END_IF
	END_IF


4: 	(* UA_Read *)
	fbUA_Read(
		Execute			:= TRUE,
		ConnectionHdl	:= nConnectionHdl,
		NodeHdl			:= nNodeHdl,
		stNodeAddInfo 	:= stNodeAddInfo,
		cbData			:= GVL_ArrayTests2DimPLC.NodeID_Sizes[nLoopVars], //SIZEOF(nReadData),		
		pVariable		:= ADR(GVL_ArrayTests2DimPLC.NodeID_ReadWrittenResults[nLoopVars].nData) //Variable
		);

	IF NOT fbUA_Read.Busy THEN
		fbUA_Read(
			Execute 	:= FALSE);

		IF NOT fbUA_Read.Error THEN
			(* session closed *)
			iState 		:= iState + 1; (* idle *)
			a := GVL_ArrayTests2DimPLC.NodeID_WriteCommands[nLoopVars].nData;
			b := GVL_ArrayTests2DimPLC.NodeID_ReadWrittenResults[nLoopVars].nData;
			FOR counter:=1 TO fbUA_Read.cbData_R //fbUA_Read.GVL_ScalarTests.NodeID_Sizes[nLoopVars]
			DO
				a_ := a[counter];
				b_ := b[counter];
				IF(NOT a_ = b_) THEN
					EXIT;
				END_IF
			END_FOR
			IF(Counter = fbUA_Read.cbData_R+1) THEN //GVL_ScalarTests.NodeID_Sizes[nLoopVars]+1) THEN //all bytes are equal as long as length site is defined
				GVL_ArrayTests2DimPLC.NodeID_CheckReadWrite[nLoopVars] := TRUE;
			END_IF 
			//Do we need this? We simply store in UNION! MEMCPY(ADR(nReadData),ADR(Variable),SIZEOF(nReadData));
		ELSE
			bError		:= TRUE;
			nErrorID	:= fbUA_Read.ErrorID;
			iState 		:= 7; (* idle *)
		END_IF
	END_IF



5:	(* Release Node Handle *)
	fbUA_NodeReleaseHandle(
		Execute			:= TRUE,
		ConnectionHdl	:= nConnectionHdl,
		NodeHdl			:= nNodeHdl
	);

	IF NOT fbUA_NodeReleaseHandle.Busy THEN
		fbUA_NodeReleaseHandle(Execute := FALSE);

		IF NOT fbUA_NodeReleaseHandle.Error THEN
			(* session closed *)
			iState 		:= iState + 1; (* idle *)
		ELSE
			bError		:= TRUE;
			nErrorID	:= fbUA_NodeReleaseHandle.ErrorID;
			iState 		:= 6; (* idle *)
		END_IF
	END_IF


6:	(* close session *)
	fbUA_Disconnect(
		Execute			:= TRUE,
		ConnectionHdl	:= nConnectionHdl
	);

	IF NOT fbUA_Disconnect.Busy THEN
		fbUA_Disconnect(Execute := FALSE);

		IF NOT fbUA_Disconnect.Error THEN
			(* session closed *)
			iState 		:= 0; (* idle *)
			//restart with next var, if existing in array
			IF(nLoopVars < nEndOfNodeIDVarsArray_2Dim) THEN
				nLoopVars := nLoopVars+1;
				bTest := TRUE;
			ELSE 
				bBusy 		:= FALSE;
				//prepare for next call 
				bTest := TRUE;
				nLoopVars := 0;
			END_IF
		ELSE
			bError			:= TRUE;
			nErrorID		:= fbUA_Disconnect.ErrorID;
			iState 			:= 0; (* idle *)
			nConnectionHdl	:= 0;
		END_IF
	END_IF
END_CASE

END_PROGRAM

// ---- Tests_Henning/POUs/PRG_3DArrayTest.TcPOU
PROGRAM PRG_3DArrayTest
VAR
	iState: INT := 3; //we need to wait for UAServer to provide variables
END_VAR

CASE iState OF
0:	
	PRG_3DArrayTest_Read();
	IF(NOT PRG_3DArrayTest_Read.bBusy AND NOT PRG_3DArrayTest_Read.bError) THEN
		iState := iState+1;
	END_IF
1:
	PRG_3DArrayTest_Write();
	IF(NOT PRG_3DArrayTest_Write.bBusy AND NOT PRG_3DArrayTest_Write.bError) THEN
		iState := iState+1;
	END_IF
2:
	PRG_3DArrayTest_ReadWritten();
	IF(NOT PRG_3DArrayTest_ReadWritten.bBusy AND NOT PRG_3DArrayTest_ReadWritten.bError) THEN
		iState := iState+1;
	END_IF
END_CASE

END_PROGRAM

// ---- Tests_Henning/POUs/PRG_3DArrayTest_Read.TcPOU
PROGRAM PRG_3DArrayTest_Read
VAR
	fbUA_Connect: UA_Connect;
	SessionConnectInfo: ST_UASessionConnectInfo;
	nConnectionHdl: DWORD;
	fbUA_GetNamespaceIndex: UA_GetNamespaceIndex;
	nNamespaceIndex: UINT;
	fbUA_NodeGetHandle: UA_NodeGetHandle;
	NodeID: ST_UANodeID;
	nNodeHdl: DWORD;
	fbUA_Read: UA_Read;
	stIndexRange: ARRAY[1..nMaxIndexRange] OF ST_UAIndexRange;
	nIndexRangeCount: UINT;
	stNodeAddInfo: ST_UANodeAdditionalInfo;
	Variable: ARRAY[1..nMaxReadDataArray_3Dim] OF BYTE;
	///DINT; 		// change the data type according to the variable type to be read
	nReadData: STRING;
	fbUA_NodeReleaseHandle: UA_NodeReleaseHandle;
	fbUA_Disconnect: UA_Disconnect;
	iState: INT;
	bTest: BOOL := TRUE;
	bDone: BOOL;
	bBusy: BOOL;
	bError: BOOL;
	nErrorID: DWORD;
	nLoopVars: UINT;
END_VAR

CASE iState OF
0:	(* idle *)
	IF bTest THEN
		bTest		:= FALSE;
		bError		:= FALSE;
		nErrorID	:= 0;
		bBusy 		:= TRUE; 
		SessionConnectInfo.tConnectTimeout 		:= T#9S;
		SessionConnectInfo.tSessionTimeout 		:= T#9S;
		SessionConnectInfo.sApplicationName		:= '';
		SessionConnectInfo.sApplicationUri 		:= '';
		SessionConnectInfo.eSecurityMode 		:= eUASecurityMsgMode_None;
		SessionConnectInfo.eSecurityPolicyUri 	:= eUASecurityPolicy_None;
		SessionConnectInfo.eTransportProfileUri := eUATransportProfileUri_UATcp;

		stNodeAddInfo.nIndexRangeCount := nIndexRangeCount;
		stNodeAddInfo.stIndexRange := stIndexRange;
		iState	:= iState + 1;
	END_IF

1:	(* open UA session *)
	fbUA_Connect(
		Execute				:= TRUE,
		ServerURL			:= GVL_ArrayTests3DimPLC.sOpcUA_URL,
		SessionConnectInfo	:= SessionConnectInfo,
		Timeout				:= T#10S,
		ConnectionHdl		=> nConnectionHdl
	);

	IF NOT fbUA_Connect.Busy THEN
		fbUA_Connect(Execute := FALSE);

		IF NOT fbUA_Connect.Error THEN
			(* session open *)
			iState := iState + 1;
		ELSE
			bError			:= TRUE;
			nErrorID		:= fbUA_Connect.ErrorID;
			nConnectionHdl	:= 0;
			iState 			:= 0; (* idle *)
		END_IF
	END_IF


2:	(* GetNS Index *)
	IF NOT GVL_ArrayTests3DimPLC.NodeID_DoOrDont[nLoopVars] THEN
		iState := 6;
	END_IF
	fbUA_GetNamespaceIndex(
		Execute			:= TRUE,
		ConnectionHdl	:= nConnectionHdl,
		NamespaceUri	:= GVL_ArrayTests3DimPLC.sNodeIDNamespace,
		NamespaceIndex	=> nNamespaceIndex
	);

	IF NOT fbUA_GetNamespaceIndex.Busy THEN
		fbUA_GetNamespaceIndex(Execute := FALSE);

		IF NOT fbUA_GetNamespaceIndex.Error THEN
			(* session closed *)
			iState 		:= iState + 1; (* idle *)
		ELSE
			bError		:= TRUE;
			nErrorID	:= fbUA_GetNamespaceIndex.ErrorID;
			iState 		:= 6; (* idle *)
		END_IF
	END_IF


3:	(* Get Node Handle *)
	NodeID.eIdentifierType := eUAIdentifierType_String;
	NodeID.nNamespaceIndex := nNamespaceIndex;
	NodeID.sIdentifier	:= GVL_ArrayTests3DimPLC.NodeID_Identifiers[nLoopVars]; // 'GVL_static.stat_BSTR_0';
	fbUA_NodeGetHandle(
		Execute			:= TRUE,
		ConnectionHdl	:= nConnectionHdl,
		NodeID			:= NodeID,
		NodeHdl			=> nNodeHdl
	);

	IF NOT fbUA_NodeGetHandle.Busy THEN
		fbUA_NodeGetHandle(Execute := FALSE);

		IF NOT fbUA_NodeGetHandle.Error THEN
			(* session closed *)
			iState 		:= iState + 1; (* idle *)
		ELSE
			bError		:= TRUE;
			nErrorID	:= fbUA_NodeGetHandle.ErrorID;
			iState 		:= 6; (* idle *)
		END_IF
	END_IF


4: 	(* UA_Read *)
	fbUA_Read(
		Execute			:= TRUE,
		ConnectionHdl	:= nConnectionHdl,
		NodeHdl			:= nNodeHdl,
		stNodeAddInfo 	:= stNodeAddInfo,
		cbData			:= GVL_ArrayTests3DimPLC.NodeID_Sizes[nLoopVars], //SIZEOF(nReadData),
		pVariable		:= ADR(GVL_ArrayTests3DimPLC.NodeID_ReadResults[nLoopVars].nData) //Variable
		);

	IF NOT fbUA_Read.Busy THEN
		fbUA_Read(
			Execute 	:= FALSE);

		IF NOT fbUA_Read.Error THEN
			(* session closed *)
			iState 		:= iState + 1; (* idle *)
			//Do we need this? We simply store in UNION! MEMCPY(ADR(nReadData),ADR(Variable),SIZEOF(nReadData));
		ELSE
			bError		:= TRUE;
			nErrorID	:= fbUA_Read.ErrorID;
			iState 		:= 7; (* idle *)
		END_IF
	END_IF



5:	(* Release Node Handle *)
	fbUA_NodeReleaseHandle(
		Execute			:= TRUE,
		ConnectionHdl	:= nConnectionHdl,
		NodeHdl			:= nNodeHdl
	);

	IF NOT fbUA_NodeReleaseHandle.Busy THEN
		fbUA_NodeReleaseHandle(Execute := FALSE);

		IF NOT fbUA_NodeReleaseHandle.Error THEN
			(* session closed *)
			iState 		:= iState + 1; (* idle *)
		ELSE
			bError		:= TRUE;
			nErrorID	:= fbUA_NodeReleaseHandle.ErrorID;
			iState 		:= 6; (* idle *)
		END_IF
	END_IF


6:	(* close session *)
	fbUA_Disconnect(
		Execute			:= TRUE,
		ConnectionHdl	:= nConnectionHdl
	);

	IF NOT fbUA_Disconnect.Busy THEN
		fbUA_Disconnect(Execute := FALSE);

		IF NOT fbUA_Disconnect.Error THEN
			(* session closed *)
			iState 		:= 0; (* idle *)
			//restart with next var, if existing in array
			IF(nLoopVars < nEndOfNodeIDVarsArray_3Dim) THEN
				nLoopVars := nLoopVars+1;
				bTest := TRUE;
			ELSE 
				bBusy 		:= FALSE;
				//prepare for next call 
				bTest := TRUE;
				nLoopVars := 0;
			END_IF
		ELSE
			bError			:= TRUE;
			nErrorID		:= fbUA_Disconnect.ErrorID;
			iState 			:= 0; (* idle *)
			nConnectionHdl	:= 0;
		END_IF
	END_IF
END_CASE

END_PROGRAM

// ---- Tests_Henning/POUs/PRG_3DArrayTest_Write.TcPOU
PROGRAM PRG_3DArrayTest_Write
VAR
	fbUA_Connect: UA_Connect;
	SessionConnectInfo: ST_UASessionConnectInfo;
	sOpcUA_URL: STRING(MAX_STRING_LENGTH);
	nConnectionHdl: DWORD;
	fbUA_GetNamespaceIndex: UA_GetNamespaceIndex;
	sNamespaceUri: STRING(MAX_STRING_LENGTH);
	nNamespaceIndex: UINT;
	fbUA_NodeGetHandle: UA_NodeGetHandle;
	NodeID: ST_UANodeID;
	nNodeHdl: DWORD;
	fbUA_Write: UA_Write;
	stIndexRange: ARRAY[1..nMaxIndexRange] OF ST_UAIndexRange;
	nIndexRangeCount: UINT;
	stNodeAddInfo: ST_UANodeAdditionalInfo;
	/// UDINT := 12312345;		// change according to the type of variable
	nWriteData: STRING := 'Hallo';
	Variable: ARRAY[1..nMaxReadData] OF BYTE;
	cbData: UDINT;
	fbUA_NodeReleaseHandle: UA_NodeReleaseHandle;
	fbUA_Disconnect: UA_Disconnect;
	iState: INT;
	bTest: BOOL := TRUE;
	bDone: BOOL;
	bBusy: BOOL;
	bError: BOOL;
	nErrorID: DWORD;
	nLoopVars: UINT;
END_VAR

CASE iState OF
0:	(* idle *)
	IF bTest THEN
		bTest	:= FALSE;
		bError	:= FALSE;
		nErrorID	:= 0;
		bBusy := TRUE; 

		(* Parameterize 
		GVL_ScalarTests.NodeID_WriteCommands[0].bBool := TRUE; 
		GVL_ScalarTests.NodeID_WriteCommands[1].sString := 'WriteTest'; 
		GVL_ScalarTests.NodeID_WriteCommands[2].bByte := 123; 
		GVL_ScalarTests.NodeID_WriteCommands[3].nInt := 124; 
		GVL_ScalarTests.NodeID_WriteCommands[4].nUdint := 125; 
		GVL_ScalarTests.NodeID_WriteCommands[5].nLReal := 1.23456; //R8x 
		GVL_ScalarTests.NodeID_WriteCommands[6].bByte := 111; 
		GVL_ScalarTests.NodeID_WriteCommands[7].nInt := 112; 
		GVL_ScalarTests.NodeID_WriteCommands[8].nUdint := 113; 
		*)
		
		SessionConnectInfo.tConnectTimeout 		:= T#9S;
		SessionConnectInfo.tSessionTimeout 		:= T#9S;
		SessionConnectInfo.sApplicationName		:= '';
		SessionConnectInfo.sApplicationUri 		:= '';
		SessionConnectInfo.eSecurityMode 		:= eUASecurityMsgMode_None;
		SessionConnectInfo.eSecurityPolicyUri 	:= eUASecurityPolicy_None;
		SessionConnectInfo.eTransportProfileUri := eUATransportProfileUri_UATcp;
		
		stNodeAddInfo.nIndexRangeCount := nIndexRangeCount;
		stNodeAddInfo.stIndexRange := stIndexRange;
		iState	:= iState + 1;
	END_IF

1:	(* open UA session *)
	fbUA_Connect(
		Execute				:= TRUE,
		ServerURL			:= GVL_ArrayTests3DimPLC.sOpcUA_URL,
		SessionConnectInfo	:= SessionConnectInfo,
		Timeout				:= T#10S,
		ConnectionHdl		=> nConnectionHdl
	);

	IF NOT fbUA_Connect.Busy THEN
		fbUA_Connect(Execute := FALSE);

		IF NOT fbUA_Connect.Error THEN
			(* session open *)
			iState := iState + 1;
		ELSE
			bError			:= TRUE;
			nErrorID		:= fbUA_Connect.ErrorID;
			nConnectionHdl	:= 0;
			iState 			:= 0; (* idle *)
		END_IF
	END_IF


2:	(* GetNS Index *)
	IF NOT GVL_ArrayTests3DimPLC.NodeID_DoOrDont[nLoopVars] THEN
		iState := 6;
	END_IF
	fbUA_GetNamespaceIndex(
		Execute			:= TRUE,
		ConnectionHdl	:= nConnectionHdl,
		NamespaceUri	:= GVL_ArrayTests3DimPLC.sNodeIDNamespace,
		NamespaceIndex	=> nNamespaceIndex
	);

	IF NOT fbUA_GetNamespaceIndex.Busy THEN
		fbUA_GetNamespaceIndex(Execute := FALSE);

		IF NOT fbUA_GetNamespaceIndex.Error THEN
			(* session closed *)
			iState 		:= iState + 1; (* idle *)
		ELSE
			bError		:= TRUE;
			nErrorID	:= fbUA_GetNamespaceIndex.ErrorID;
			iState 		:= 6; (* idle *)
		END_IF
	END_IF


3:	(* Get Node Handle *)
	NodeID.eIdentifierType := eUAIdentifierType_String;
	NodeID.nNamespaceIndex := nNamespaceIndex;
	NodeID.sIdentifier	:= GVL_ArrayTests3DimPLC.NodeID_Identifiers[nLoopVars]; // 'GVL_static.stat_BSTR_0';
	fbUA_NodeGetHandle(
		Execute			:= TRUE,
		ConnectionHdl	:= nConnectionHdl,
		NodeID			:= NodeID,
		NodeHdl			=> nNodeHdl
	);

	IF NOT fbUA_NodeGetHandle.Busy THEN
		fbUA_NodeGetHandle(Execute := FALSE);

		IF NOT fbUA_NodeGetHandle.Error THEN
			(* session closed *)
			IF SIZEOF(nWriteData) <= nMaxReadData THEN 
				iState 		:= iState + 1; (* idle *)
				MEMSET(ADR(Variable),0,SIZEOF(Variable));
				MEMCPY(ADR(Variable),ADR(nWriteData),SIZEOF(nWriteData));
			ELSE
				//cannot write buffer too small -> increase the value of nMaxData in GVL
				bError		:= TRUE;
				iState 		:= 6; (* idle *)
			END_IF
		ELSE
			bError		:= TRUE;
			nErrorID	:= fbUA_NodeGetHandle.ErrorID;
			iState 		:= 6; (* idle *)
		END_IF
	END_IF


4: 	(* UA_Write *)
	fbUA_Write(
		Execute			:= TRUE,
		ConnectionHdl	:= nConnectionHdl,
		NodeHdl			:= nNodeHdl,
		stNodeAddInfo	:= stNodeAddInfo,
		cbData			:= GVL_ArrayTests3DimPLC.NodeID_Sizes[nLoopVars], //SIZEOF(nWriteData),
		pVariable		:= ADR(GVL_ArrayTests3DimPLC.NodeID_WriteCommands[nLoopVars].nData) // Variable		:= Variable
		);

	IF NOT fbUA_Write.Busy THEN
		fbUA_Write(
			Execute 		:= FALSE);

		IF NOT fbUA_Write.Error THEN
			(* session closed *)
			iState 		:= iState + 1; (* idle *)
		ELSE
			bError		:= TRUE;
			nErrorID	:= fbUA_Write.ErrorID;
			iState 		:= 7; (* idle *)
		END_IF
	END_IF


5:	(* Release Node Handle *)
	fbUA_NodeReleaseHandle(
		Execute			:= TRUE,
		ConnectionHdl	:= nConnectionHdl,
		NodeHdl			:= nNodeHdl
	);

	IF NOT fbUA_NodeReleaseHandle.Busy THEN
		fbUA_NodeReleaseHandle(Execute := FALSE);

		IF NOT fbUA_NodeReleaseHandle.Error THEN
			(* session closed *)
			iState 		:= iState + 1; (* idle *)
		ELSE
			bError		:= TRUE;
			nErrorID	:= fbUA_NodeReleaseHandle.ErrorID;
			iState 		:= 6; (* idle *)
		END_IF
	END_IF


6:	(* close session *)
	fbUA_Disconnect(
		Execute			:= TRUE,
		ConnectionHdl	:= nConnectionHdl
	);

	IF NOT fbUA_Disconnect.Busy THEN
		fbUA_Disconnect(Execute := FALSE);

		IF NOT fbUA_Disconnect.Error THEN
			(* session closed *)
			iState 		:= 0; (* idle *)			//restart with next var, if existing in array
			IF(nLoopVars < nEndOfNodeIDVarsArray_3Dim) THEN
				nLoopVars := nLoopVars+1;
				bTest := TRUE;
			ELSE 
				bBusy 		:= FALSE;
				//prepare for next call
				bTest := TRUE; 
				nLoopVars := 0;
			END_IF
		ELSE
			bError		:= TRUE;
			nErrorID	:= fbUA_Disconnect.ErrorID;
			iState 		:= 0; (* idle *)
			nConnectionHdl	:= 0;
		END_IF
	END_IF
END_CASE

END_PROGRAM

// ---- Tests_Henning/POUs/PRG_3DArrayTest_ReadWritten.TcPOU
PROGRAM PRG_3DArrayTest_ReadWritten
VAR
	fbUA_Connect: UA_Connect;
	SessionConnectInfo: ST_UASessionConnectInfo;
	nConnectionHdl: DWORD;
	fbUA_GetNamespaceIndex: UA_GetNamespaceIndex;
	nNamespaceIndex: UINT;
	fbUA_NodeGetHandle: UA_NodeGetHandle;
	NodeID: ST_UANodeID;
	nNodeHdl: DWORD;
	fbUA_Read: UA_Read;
	stIndexRange: ARRAY[1..nMaxIndexRange] OF ST_UAIndexRange;
	nIndexRangeCount: UINT;
	stNodeAddInfo: ST_UANodeAdditionalInfo;
	Variable: ARRAY[1..nMaxReadData] OF BYTE;
	///DINT; 		// change the data type according to the variable type to be read
	nReadData: STRING;
	fbUA_NodeReleaseHandle: UA_NodeReleaseHandle;
	fbUA_Disconnect: UA_Disconnect;
	iState: INT;
	bTest: BOOL := TRUE;
	bDone: BOOL;
	bBusy: BOOL;
	bError: BOOL;
	nErrorID: DWORD;
	nLoopVars: UINT;
	counter: UDINT;
	a: ARRAY[1..nMaxReadDataArray_3Dim] OF BYTE;
	b: ARRAY[1..nMaxReadDataArray_3Dim] OF BYTE;
	a_: BYTE;
	b_: BYTE;
	nTmpL: UINT;
END_VAR

CASE iState OF
0:	(* idle *)
	IF bTest THEN
		bTest		:= FALSE;
		bError		:= FALSE;
		nErrorID	:= 0;
		bBusy 		:= TRUE; 
		SessionConnectInfo.tConnectTimeout 		:= T#9S;
		SessionConnectInfo.tSessionTimeout 		:= T#9S;
		SessionConnectInfo.sApplicationName		:= '';
		SessionConnectInfo.sApplicationUri 		:= '';
		SessionConnectInfo.eSecurityMode 		:= eUASecurityMsgMode_None;
		SessionConnectInfo.eSecurityPolicyUri 	:= eUASecurityPolicy_None;
		SessionConnectInfo.eTransportProfileUri := eUATransportProfileUri_UATcp;

		stNodeAddInfo.nIndexRangeCount := nIndexRangeCount;
		stNodeAddInfo.stIndexRange := stIndexRange;
		iState	:= iState + 1;
	END_IF

1:	(* open UA session *)
	fbUA_Connect(
		Execute				:= TRUE,
		ServerURL			:= GVL_ArrayTests3DimPLC.sOpcUA_URL,
		SessionConnectInfo	:= SessionConnectInfo,
		Timeout				:= T#10S,
		ConnectionHdl		=> nConnectionHdl
	);

	IF NOT fbUA_Connect.Busy THEN
		fbUA_Connect(Execute := FALSE);

		IF NOT fbUA_Connect.Error THEN
			(* session open *)
			iState := iState + 1;
		ELSE
			bError			:= TRUE;
			nErrorID		:= fbUA_Connect.ErrorID;
			nConnectionHdl	:= 0;
			iState 			:= 0; (* idle *)
		END_IF
	END_IF


2:	(* GetNS Index *)
	IF NOT GVL_ArrayTests3DimPLC.NodeID_DoOrDont[nLoopVars] THEN
		iState := 6;
	END_IF
	fbUA_GetNamespaceIndex(
		Execute			:= TRUE,
		ConnectionHdl	:= nConnectionHdl,
		NamespaceUri	:= GVL_ArrayTests3DimPLC.sNodeIDNamespace,
		NamespaceIndex	=> nNamespaceIndex
	);

	IF NOT fbUA_GetNamespaceIndex.Busy THEN
		fbUA_GetNamespaceIndex(Execute := FALSE);

		IF NOT fbUA_GetNamespaceIndex.Error THEN
			(* session closed *)
			iState 		:= iState + 1; (* idle *)
		ELSE
			bError		:= TRUE;
			nErrorID	:= fbUA_GetNamespaceIndex.ErrorID;
			iState 		:= 6; (* idle *)
		END_IF
	END_IF


3:	(* Get Node Handle *)
	NodeID.eIdentifierType := eUAIdentifierType_String;
	NodeID.nNamespaceIndex := nNamespaceIndex;
	NodeID.sIdentifier	:= GVL_ArrayTests3DimPLC.NodeID_Identifiers[nLoopVars]; // 'GVL_static.stat_BSTR_0';
	fbUA_NodeGetHandle(
		Execute			:= TRUE,
		ConnectionHdl	:= nConnectionHdl,
		NodeID			:= NodeID,
		NodeHdl			=> nNodeHdl
	);

	IF NOT fbUA_NodeGetHandle.Busy THEN
		fbUA_NodeGetHandle(Execute := FALSE);

		IF NOT fbUA_NodeGetHandle.Error THEN
			(* session closed *)
			iState 		:= iState + 1; (* idle *)
		ELSE
			bError		:= TRUE;
			nErrorID	:= fbUA_NodeGetHandle.ErrorID;
			iState 		:= 6; (* idle *)
		END_IF
	END_IF


4: 	(* UA_Read *)
	fbUA_Read(
		Execute			:= TRUE,
		ConnectionHdl	:= nConnectionHdl,
		NodeHdl			:= nNodeHdl,
		stNodeAddInfo 	:= stNodeAddInfo,
		cbData			:= GVL_ArrayTests3DimPLC.NodeID_Sizes[nLoopVars], //SIZEOF(nReadData),		
		pVariable		:= ADR(GVL_ArrayTests3DimPLC.NodeID_ReadWrittenResults[nLoopVars].nData) //Variable
		);

	IF NOT fbUA_Read.Busy THEN
		fbUA_Read(
			Execute 	:= FALSE);

		IF NOT fbUA_Read.Error THEN
			(* session closed *)
			iState 		:= iState + 1; (* idle *)
			a := GVL_ArrayTests3DimPLC.NodeID_WriteCommands[nLoopVars].nData;
			b := GVL_ArrayTests3DimPLC.NodeID_ReadWrittenResults[nLoopVars].nData;
			FOR counter:=1 TO fbUA_Read.cbData_R //fbUA_Read.GVL_ScalarTests.NodeID_Sizes[nLoopVars]
			DO
				a_ := a[counter];
				b_ := b[counter];
				IF(NOT a_ = b_) THEN
					EXIT;
				END_IF
			END_FOR
			IF(Counter = fbUA_Read.cbData_R+1) THEN //GVL_ScalarTests.NodeID_Sizes[nLoopVars]+1) THEN //all bytes are equal as long as length site is defined
				GVL_ArrayTests3DimPLC.NodeID_CheckReadWrite[nLoopVars] := TRUE;
			END_IF 
			//Do we need this? We simply store in UNION! MEMCPY(ADR(nReadData),ADR(Variable),SIZEOF(nReadData));
		ELSE
			bError		:= TRUE;
			nErrorID	:= fbUA_Read.ErrorID;
			iState 		:= 7; (* idle *)
		END_IF
	END_IF



5:	(* Release Node Handle *)
	fbUA_NodeReleaseHandle(
		Execute			:= TRUE,
		ConnectionHdl	:= nConnectionHdl,
		NodeHdl			:= nNodeHdl
	);

	IF NOT fbUA_NodeReleaseHandle.Busy THEN
		fbUA_NodeReleaseHandle(Execute := FALSE);

		IF NOT fbUA_NodeReleaseHandle.Error THEN
			(* session closed *)
			iState 		:= iState + 1; (* idle *)
		ELSE
			bError		:= TRUE;
			nErrorID	:= fbUA_NodeReleaseHandle.ErrorID;
			iState 		:= 6; (* idle *)
		END_IF
	END_IF


6:	(* close session *)
	fbUA_Disconnect(
		Execute			:= TRUE,
		ConnectionHdl	:= nConnectionHdl
	);

	IF NOT fbUA_Disconnect.Busy THEN
		fbUA_Disconnect(Execute := FALSE);

		IF NOT fbUA_Disconnect.Error THEN
			(* session closed *)
			iState 		:= 0; (* idle *)
			//restart with next var, if existing in array
			IF(nLoopVars < nEndOfNodeIDVarsArray_3Dim) THEN
				nLoopVars := nLoopVars+1;
				bTest := TRUE;
			ELSE 
				bBusy 		:= FALSE;
				//prepare for next call 
				bTest := TRUE;
				nLoopVars := 0;
			END_IF
		ELSE
			bError			:= TRUE;
			nErrorID		:= fbUA_Disconnect.ErrorID;
			iState 			:= 0; (* idle *)
			nConnectionHdl	:= 0;
		END_IF
	END_IF
END_CASE

END_PROGRAM

// ---- Tests_Henning/POUs/PRG_Connect_Encrypted.TcPOU
PROGRAM PRG_Connect_Encrypted
VAR
	fbUA_Connect			: UA_Connect;
	SessionConnectInfo		: ST_UASessionConnectInfo;
	sOpcUA_URL				: STRING(MAX_STRING_LENGTH);
	nConnectionHdl			: DWORD;

	fbUA_GetNamespaceIndex 	: UA_GetNamespaceIndex;
	nNamespaceIndex			: UINT := -1;

	fbUA_NodeGetHandle		: UA_NodeGetHandle;
	NodeID					: ST_UANodeID;
	nNodeHdl				: DWORD;

	fbUA_Read				: UA_Read;
	stIndexRange			: ARRAY [1..nMaxIndexRange] OF ST_UAIndexRange;
	nIndexRangeCount		: UINT;
	stNodeAddInfo			: ST_UANodeAdditionalInfo;
	nReadData				: DINT; 		// change the data type according to the variable type to be read
	bReadData				: DINT; 
	sReadData				: STRING(4);
	cbData_R				: UDINT;
	
	fbUA_NodeReleaseHandle	: UA_NodeReleaseHandle;

	fbUA_Disconnect		: UA_Disconnect;

	iState		: INT;
	bTest		: BOOL:= TRUE;
	bDone		: BOOL;
	bBusy		: BOOL;
	bError		: BOOL;
	nErrorID	: DWORD;
END_VAR

//Connect Encryped with the demoserver
//Certs of demoserver (due to serverconfig.xml) are located: C:\ProgramData\UnifiedAutomation\UaSdkCppBundleSource/pkiserver/
//just retrieves nNamespaceIndex from http://opcfoundation.org/UA/ - should be 0 (init of nNamespaceIndex := -1)

CASE iState OF
0:	(* idle *)
	IF bTest THEN
		bTest		:= FALSE;
		bDone 		:= FALSE; 
		bError		:= FALSE;
		nErrorID	:= 0;
		nNamespaceIndex := -1;
		
		(* Parameterize *)
		sOpcUA_URL						:= 'opc.tcp://localhost:48010';	(* OpcUA Url of the device with ip address *)

		SessionConnectInfo.tConnectTimeout 		:= T#1M;
		SessionConnectInfo.tSessionTimeout 		:= T#1M;
		SessionConnectInfo.sApplicationName		:= '';
		SessionConnectInfo.sApplicationUri 		:= 'HENNINGM-NB';
		SessionConnectInfo.eSecurityMode 		:= eUASecurityMsgMode_Sign_Encrypt;
		SessionConnectInfo.eSecurityPolicyUri 	:= eUASecurityPolicy_Basic128Rsa15;
		SessionConnectInfo.eTransportProfileUri := eUATransportProfileUri_UATcp;

(*		nIndexRange[1].nStartIndex := 0;
		nIndexRange[1].nEndIndex := 1;
		nIndexRange[1].bRangeAccess := TRUE; *)
		stNodeAddInfo.nIndexRangeCount := nIndexRangeCount;
		stNodeAddInfo.stIndexRange := stIndexRange;
		iState	:= iState + 1;
	END_IF

1:	(* open UA session *)
	fbUA_Connect(
		Execute				:= TRUE,
		ServerURL			:= sOpcUA_URL,
		SessionConnectInfo	:= SessionConnectInfo,
		Timeout				:= T#5S,
		ConnectionHdl		=> nConnectionHdl
	);

	IF NOT fbUA_Connect.Busy THEN
		fbUA_Connect(Execute := FALSE);

		IF NOT fbUA_Connect.Error THEN
			(* session open *)
			iState := iState + 1;
		ELSE
			bError			:= TRUE;
			nErrorID		:= fbUA_Connect.ErrorID;
			nConnectionHdl	:= 0;
			iState 			:= 0; (* idle *)
		END_IF
	END_IF


2:	(* GetNS Index *)
	fbUA_GetNamespaceIndex(
		Execute			:= TRUE,
		ConnectionHdl	:= nConnectionHdl,
		//NamespaceUri	:= 'PLC1', 
		NamespaceUri	:= 'http://opcfoundation.org/UA/',
		NamespaceIndex	=> nNamespaceIndex
	);

	IF NOT fbUA_GetNamespaceIndex.Busy THEN
		fbUA_GetNamespaceIndex(Execute := FALSE);
		IF NOT fbUA_GetNamespaceIndex.Error THEN
			(* session closed *)
			iState 		:= iState + 6; (* idle *)
			bDone := TRUE; 
		ELSE
			bError		:= TRUE;
			nErrorID	:= fbUA_GetNamespaceIndex.ErrorID;
			iState 		:= 6; (* idle *)
		END_IF
	END_IF


6:	(* close session *)
	fbUA_Disconnect(
		Execute			:= TRUE,
		ConnectionHdl	:= nConnectionHdl
	);

	IF NOT fbUA_Disconnect.Busy THEN
		fbUA_Disconnect(Execute := FALSE);
		bBusy := FALSE;
		IF NOT fbUA_Disconnect.Error THEN
			(* session closed *)
			iState 		:= 0; (* idle *)
			IF NOT bError THEN 
				bDone 	:= TRUE;
			END_IF
		ELSE
			bError			:= TRUE;
			nErrorID		:= fbUA_Disconnect.ErrorID;
			iState 			:= 0; (* idle *)
			nConnectionHdl	:= 0;
		END_IF
	END_IF
END_CASE

END_PROGRAM

// ---- Tests_Henning/POUs/PRG_GetBrokenHandle.TcPOU
PROGRAM PRG_GetBrokenHandle
VAR
	fbUA_Connect			: UA_Connect;
	SessionConnectInfo		: ST_UASessionConnectInfo;
	sOpcUA_URL				: STRING(MAX_STRING_LENGTH);
	nConnectionHdl			: DWORD;

	fbUA_GetNamespaceIndex 	: UA_GetNamespaceIndex;
	nNamespaceIndex			: UINT;

	fbUA_NodeGetHandle		: UA_NodeGetHandle;
	NodeID					: ST_UANodeID;
	nNodeHdl				: DWORD;

	fbUA_Read				: UA_Read;
	stIndexRange			: ARRAY [1..nMaxIndexRange] OF ST_UAIndexRange;
	nIndexRangeCount		: UINT;
	stNodeAddInfo			: ST_UANodeAdditionalInfo;
	nReadData				: DINT; 		// change the data type according to the variable type to be read
	bReadData				: DINT; 
	sReadData				: STRING(4);
	cbData_R				: UDINT;
	
	fbUA_NodeReleaseHandle	: UA_NodeReleaseHandle;

	fbUA_Disconnect		: UA_Disconnect;

	iState		: INT;
	bTest		: BOOL:= TRUE;
	bDone		: BOOL;
	bTestSuccessfull : BOOL;
	bBusy		: BOOL;
	bError		: BOOL;
	nErrorID	: DWORD;
END_VAR

// FALSE-Test!!! Check bTestSuccessfull for Success !!!
// This should fail.
// Simulates access to a nodeid with wrong arraydim vs valuerank information.
// FALSE-Test!!! Check bTestSuccessfull for Success !!!

CASE iState OF
0:	(* idle *)
	IF bTest THEN
		bTest		:= FALSE;
		bError		:= FALSE;
		nErrorID	:= 0;

		(* Parameterize *)
		sOpcUA_URL						:= 'opc.tcp://henningm-nb:4841';	(* OpcUA Url of the device with ip address *)

		SessionConnectInfo.tConnectTimeout 		:= T#1M;
		SessionConnectInfo.tSessionTimeout 		:= T#1M;
		SessionConnectInfo.sApplicationName		:= '';
		SessionConnectInfo.sApplicationUri 		:= '';
		SessionConnectInfo.eSecurityMode 		:= eUASecurityMsgMode_None;
		SessionConnectInfo.eSecurityPolicyUri 	:= eUASecurityPolicy_None;
		SessionConnectInfo.eTransportProfileUri := eUATransportProfileUri_UATcp;

